C05474=1225.278,36.336,-43.631,-179.133,5.420,148.684
C05475=1225.283,36.087,-43.615,-179.135,5.420,148.685
C05476=1225.289,35.837,-43.599,-179.138,5.420,148.685
C05477=1225.293,35.588,-43.583,-179.141,5.419,148.686
C05478=1225.299,35.339,-43.567,-179.143,5.418,148.687
C05479=1225.304,35.088,-43.551,-179.146,5.418,148.687
C05480=1225.308,34.839,-43.536,-179.149,5.417,148.688
C05481=1225.313,34.591,-43.520,-179.151,5.417,148.689
C05482=1225.318,34.340,-43.504,-179.153,5.416,148.689
C05483=1225.323,34.091,-43.488,-179.156,5.416,148.690
C05484=1225.329,33.842,-43.472,-179.158,5.416,148.691
C05485=1225.333,33.592,-43.456,-179.161,5.415,148.691
C05486=1225.338,33.343,-43.441,-179.163,5.414,148.692
C05487=1225.343,33.093,-43.425,-179.166,5.414,148.693
C05488=1225.348,32.844,-43.410,-179.169,5.413,148.693
C05489=1225.353,32.595,-43.393,-179.171,5.413,148.694
C05490=1225.358,32.345,-43.377,-179.174,5.412,148.695
C05491=1225.363,32.096,-43.362,-179.176,5.413,148.695
C05492=1225.368,31.846,-43.347,-179.179,5.412,148.696
C05493=1225.373,31.596,-43.331,-179.181,5.411,148.697
C05494=1225.378,31.347,-43.314,-179.184,5.411,148.697
C05495=1225.383,31.098,-43.299,-179.186,5.410,148.698
C05496=1225.387,30.848,-43.284,-179.189,5.409,148.698
C05497=1225.393,30.599,-43.268,-179.191,5.409,148.699
C05498=1225.398,30.349,-43.252,-179.194,5.409,148.700
C05499=1225.403,30.099,-43.236,-179.196,5.409,148.701
C05500=1225.408,29.831,-43.220,-179.199,5.408,148.701
C05501=1225.413,29.563,-43.203,-179.201,5.408,148.702
C05502=1225.419,29.294,-43.186,-179.205,5.407,148.703
C05503=1225.424,29.026,-43.169,-179.207,5.407,148.703
C05504=1225.429,28.777,-43.154,-179.210,5.406,148.704
C05505=1225.434,28.526,-43.138,-179.213,5.406,148.705
C05506=1225.439,28.277,-43.122,-179.215,5.405,148.705
C05507=1225.445,28.028,-43.107,-179.217,5.404,148.706
C05508=1225.449,27.778,-43.091,-179.220,5.404,148.707
C05509=1225.454,27.528,-43.076,-179.222,5.404,148.707
C05510=1225.459,27.279,-43.060,-179.225,5.403,148.708
C05511=1225.464,27.030,-43.045,-179.227,5.403,148.709
C05512=1225.469,26.780,-43.029,-179.230,5.402,148.709
C05513=1225.474,26.530,-43.014,-179.233,5.402,148.710
C05514=1225.479,26.281,-42.999,-179.235,5.401,148.711
C05515=1225.484,26.032,-42.983,-179.237,5.401,148.711
C05516=1225.489,25.782,-42.967,-179.240,5.401,148.712
C05517=1225.494,25.533,-42.952,-179.243,5.400,148.713
C05518=1225.499,25.283,-42.937,-179.245,5.400,148.713
C05519=1225.504,25.034,-42.922,-179.248,5.399,148.714
C05520=1225.509,24.784,-42.906,-179.251,5.399,148.715
C05521=1225.514,24.535,-42.890,-179.253,5.398,148.715
C05522=1225.519,24.286,-42.875,-179.255,5.398,148.716
C05523=1225.524,24.036,-42.860,-179.257,5.398,148.717
C05524=1225.529,23.787,-42.844,-179.260,5.397,148.717
C05525=1225.533,23.537,-42.829,-179.263,5.397,148.718
C05526=1225.539,23.288,-42.813,-179.265,5.396,148.719
C05527=1225.544,23.038,-42.799,-179.268,5.395,148.719
C05528=1225.549,22.789,-42.783,-179.270,5.396,148.720
C05529=1225.553,22.539,-42.768,-179.273,5.395,148.721
C05530=1225.559,22.289,-42.752,-179.275,5.395,148.721
C05531=1225.564,22.040,-42.737,-179.278,5.394,148.722
C05532=1225.569,21.791,-42.722,-179.281,5.394,148.723
C05533=1225.574,21.541,-42.706,-179.283,5.394,148.723
C05534=1225.579,21.292,-42.691,-179.285,5.393,148.724
C05535=1225.584,21.042,-42.676,-179.288,5.393,148.725
C05536=1225.588,20.793,-42.661,-179.291,5.392,148.725
C05537=1225.594,20.543,-42.645,-179.293,5.392,148.726
C05538=1225.598,20.294,-42.630,-179.296,5.391,148.727
C05539=1225.604,20.045,-42.615,-179.298,5.391,148.727
C05540=1225.609,19.795,-42.600,-179.300,5.390,148.728
C05541=1225.614,19.545,-42.584,-179.303,5.390,148.729
C05542=1225.618,19.296,-42.569,-179.306,5.389,148.729
C05543=1225.624,19.046,-42.554,-179.308,5.389,148.730
C05544=1225.628,18.797,-42.539,-179.310,5.389,148.731
C05545=1225.634,18.547,-42.524,-179.313,5.389,148.731
C05546=1225.639,18.298,-42.509,-179.316,5.388,148.732
C05547=1225.644,18.049,-42.493,-179.318,5.388,148.733
C05548=1225.648,17.799,-42.478,-179.321,5.387,148.733
C05549=1225.654,17.549,-42.463,-179.323,5.386,148.734
C05550=1225.658,17.300,-42.448,-179.326,5.387,148.735
C05551=1225.664,17.050,-42.433,-179.328,5.386,148.735
C05552=1225.669,16.801,-42.418,-179.331,5.386,148.736
C05553=1225.674,16.551,-42.403,-179.334,5.385,148.737
C05554=1225.679,16.302,-42.388,-179.336,5.385,148.737
C05555=1225.683,16.053,-42.373,-179.338,5.385,148.738
C05556=1225.689,15.803,-42.358,-179.341,5.384,148.739
C05557=1225.693,15.553,-42.342,-179.344,5.384,148.740
C05558=1225.699,15.303,-42.328,-179.346,5.383,148.740
C05559=1225.703,15.054,-42.313,-179.349,5.383,148.741
C05560=1225.708,14.805,-42.298,-179.350,5.383,148.741
C05561=1225.714,14.555,-42.283,-179.353,5.382,148.742
C05562=1225.718,14.306,-42.268,-179.356,5.382,148.743
C05563=1225.724,14.057,-42.252,-179.358,5.381,148.743
C05564=1225.729,13.807,-42.238,-179.361,5.381,148.744
C05565=1225.733,13.558,-42.223,-179.363,5.381,148.745
C05566=1225.739,13.308,-42.208,-179.366,5.380,148.745
C05567=1225.744,13.059,-42.193,-179.368,5.380,148.746
C05568=1225.748,12.810,-42.178,-179.371,5.379,148.747
C05569=1225.754,12.560,-42.163,-179.373,5.379,148.748
C05570=1225.759,12.310,-42.148,-179.376,5.379,148.748
C05571=1225.764,12.060,-42.133,-179.378,5.378,148.749
C05572=1225.768,11.811,-42.118,-179.381,5.378,148.750
C05573=1225.773,11.561,-42.104,-179.384,5.377,148.750
C05574=1225.779,11.312,-42.088,-179.386,5.378,148.751
C05575=1225.784,11.062,-42.074,-179.388,5.377,148.752
C05576=1225.788,10.813,-42.059,-179.391,5.377,148.752
C05577=1225.793,10.563,-42.045,-179.394,5.376,148.753
C05578=1225.799,10.314,-42.029,-179.396,5.375,148.754
C05579=1225.804,10.064,-42.015,-179.398,5.376,148.754
C05580=1225.808,9.815,-42.000,-179.401,5.375,148.755
C05581=1225.814,9.565,-41.985,-179.404,5.375,148.756
C05582=1225.819,9.316,-41.970,-179.406,5.374,148.756
C05583=1225.824,9.066,-41.956,-179.408,5.374,148.757
C05584=1225.828,8.817,-41.941,-179.411,5.374,148.758
C05585=1225.834,8.567,-41.926,-179.414,5.373,148.759
C05586=1225.839,8.318,-41.911,-179.416,5.373,148.759
C05587=1225.844,8.068,-41.896,-179.418,5.373,148.760
C05588=1225.849,7.818,-41.882,-179.421,5.373,148.761
C05589=1225.854,7.569,-41.867,-179.424,5.372,148.761
C05590=1225.859,7.319,-41.852,-179.426,5.372,148.762
C05591=1225.864,7.070,-41.837,-179.429,5.371,148.762
C05592=1225.869,6.820,-41.823,-179.431,5.371,148.763
C05593=1225.874,6.570,-41.808,-179.433,5.370,148.764
C05594=1225.879,6.321,-41.793,-179.436,5.370,148.764
C05595=1225.884,6.072,-41.779,-179.439,5.369,148.765
C05596=1225.889,5.823,-41.764,-179.441,5.370,148.766
C05597=1225.894,5.574,-41.750,-179.443,5.369,148.767
C05598=1225.900,5.324,-41.735,-179.446,5.369,148.767
C05599=1225.904,5.074,-41.720,-179.449,5.368,148.768
C05600=1225.909,4.825,-41.706,-179.451,5.368,148.769
C05601=1225.914,4.575,-41.691,-179.453,5.368,148.769
C05602=1225.919,4.326,-41.677,-179.456,5.367,148.770
C05603=1225.924,4.076,-41.662,-179.459,5.367,148.771
C05604=1225.930,3.807,-41.646,-179.461,5.366,148.771
C05605=1225.935,3.538,-41.631,-179.464,5.367,148.772
C05606=1225.940,3.269,-41.615,-179.467,5.366,148.773
C05607=1225.945,3.000,-41.600,-179.469,5.366,148.774
C05608=1225.951,2.750,-41.585,-179.472,5.365,148.774
C05609=1225.956,2.501,-41.570,-179.475,5.365,148.775
C05610=1225.961,2.252,-41.556,-179.477,5.365,148.776
C05611=1225.966,2.002,-41.541,-179.479,5.365,148.776
C05612=1225.971,1.753,-41.527,-179.482,5.364,148.777
C05613=1225.976,1.503,-41.513,-179.485,5.364,148.778
C05614=1225.981,1.254,-41.498,-179.487,5.364,148.778
C05615=1225.986,1.004,-41.484,-179.489,5.363,148.779
C05616=1225.991,0.754,-41.469,-179.492,5.363,148.780
C05617=1225.996,0.505,-41.455,-179.495,5.362,148.781
C05618=1226.001,0.255,-41.440,-179.497,5.363,148.781
C05619=1226.007,0.006,-41.426,-179.499,5.362,148.782
C05620=1226.012,-0.243,-41.411,-179.502,5.362,148.783
C05621=1226.017,-0.493,-41.397,-179.505,5.361,148.783
C05622=1226.022,-0.743,-41.383,-179.507,5.361,148.784
C05623=1226.026,-0.993,-41.368,-179.509,5.361,148.785
C05624=1226.031,-1.242,-41.354,-179.512,5.360,148.785
C05625=1226.036,-1.492,-41.340,-179.515,5.360,148.786
C05626=1226.042,-1.740,-41.325,-179.517,5.360,148.787
C05627=1226.047,-1.990,-41.311,-179.519,5.359,148.787
C05628=1226.052,-2.240,-41.297,-179.522,5.359,148.788
C05629=1226.056,-2.490,-41.282,-179.525,5.358,148.789
C05630=1226.061,-2.739,-41.268,-179.527,5.359,148.789
C05631=1226.066,-2.989,-41.254,-179.529,5.358,148.790
C05632=1226.072,-3.238,-41.240,-179.532,5.358,148.791
C05633=1226.077,-3.488,-41.226,-179.534,5.358,148.792
C05634=1226.082,-3.737,-41.211,-179.537,5.357,148.792
C05635=1226.087,-3.987,-41.197,-179.539,5.357,148.793
C05636=1226.092,-4.237,-41.183,-179.542,5.356,148.794
C05637=1226.097,-4.486,-41.169,-179.544,5.357,148.794
C05638=1226.102,-4.736,-41.155,-179.547,5.356,148.795
C05639=1226.107,-4.985,-41.140,-179.550,5.356,148.796
C05640=1226.112,-5.235,-41.126,-179.552,5.355,148.796
C05641=1226.117,-5.485,-41.112,-179.554,5.355,148.797
C05642=1226.123,-5.734,-41.098,-179.557,5.355,148.798
C05643=1226.128,-5.983,-41.084,-179.560,5.354,148.798
C05644=1226.133,-6.233,-41.069,-179.562,5.355,148.799
C05645=1226.138,-6.483,-41.055,-179.564,5.354,148.800
C05646=1226.143,-6.733,-41.041,-179.567,5.354,148.801
C05647=1226.147,-6.981,-41.028,-179.570,5.353,148.801
C05648=1226.152,-7.231,-41.013,-179.572,5.353,148.802
C05649=1226.157,-7.481,-40.999,-179.574,5.353,148.803
C05650=1226.162,-7.730,-40.985,-179.577,5.352,148.803
C05651=1226.168,-7.979,-40.971,-179.579,5.353,148.804
C05652=1226.173,-8.229,-40.957,-179.582,5.352,148.805
C05653=1226.178,-8.479,-40.942,-179.584,5.352,148.805
C05654=1226.183,-8.729,-40.928,-179.587,5.351,148.806
C05655=1226.188,-8.978,-40.914,-179.589,5.352,148.807
C05656=1226.192,-9.227,-40.900,-179.592,5.351,148.807
C05657=1226.197,-9.477,-40.886,-179.594,5.350,148.808
C05658=1226.203,-9.727,-40.873,-179.597,5.351,148.809
C05659=1226.208,-9.976,-40.859,-179.599,5.350,148.810
C05660=1226.213,-10.226,-40.844,-179.602,5.350,148.810
C05661=1226.218,-10.475,-40.830,-179.604,5.350,148.811
C05662=1226.224,-10.724,-40.816,-179.607,5.350,148.812
C05663=1226.228,-10.974,-40.802,-179.609,5.349,148.812
C05664=1226.233,-11.224,-40.789,-179.612,5.349,148.813
C05665=1226.238,-11.474,-40.775,-179.614,5.349,148.814
C05666=1226.244,-11.723,-40.761,-179.617,5.348,148.814
C05667=1226.249,-11.973,-40.746,-179.619,5.348,148.815
C05668=1226.253,-12.222,-40.733,-179.621,5.348,148.816
C05669=1226.258,-12.471,-40.719,-179.624,5.348,148.816
C05670=1226.264,-12.721,-40.705,-179.627,5.347,148.817
C05671=1226.269,-12.971,-40.691,-179.629,5.347,148.818
C05672=1226.274,-13.220,-40.677,-179.631,5.347,148.819
C05673=1226.278,-13.469,-40.663,-179.634,5.346,148.819
C05674=1226.284,-13.720,-40.650,-179.637,5.346,148.820
C05675=1226.289,-13.969,-40.636,-179.639,5.346,148.821
C05676=1226.294,-14.218,-40.622,-179.641,5.346,148.821
C05677=1226.298,-14.468,-40.608,-179.644,5.345,148.822
C05678=1226.304,-14.717,-40.595,-179.646,5.345,148.823
C05679=1226.309,-14.967,-40.581,-179.649,5.345,148.823
C05680=1226.314,-15.217,-40.566,-179.651,5.344,148.824
C05681=1226.319,-15.466,-40.554,-179.654,5.345,148.825
C05682=1226.324,-15.716,-40.539,-179.656,5.344,148.825
C05683=1226.329,-15.966,-40.525,-179.659,5.344,148.826
C05684=1226.335,-16.215,-40.512,-179.661,5.344,148.827
C05685=1226.339,-16.465,-40.498,-179.664,5.343,148.828
C05686=1226.344,-16.714,-40.484,-179.666,5.343,148.828
C05687=1226.350,-16.964,-40.471,-179.668,5.343,148.829
C05688=1226.354,-17.213,-40.457,-179.671,5.343,148.830
C05689=1226.360,-17.462,-40.443,-179.674,5.342,148.830
C05690=1226.365,-17.713,-40.430,-179.676,5.342,148.831
C05691=1226.369,-17.962,-40.416,-179.678,5.342,148.832
C05692=1226.375,-18.211,-40.402,-179.681,5.342,148.832
C05693=1226.380,-18.462,-40.388,-179.684,5.341,148.833
C05694=1226.385,-18.711,-40.374,-179.686,5.341,148.834
C05695=1226.390,-18.961,-40.362,-179.688,5.341,148.834
C05696=1226.395,-19.210,-40.347,-179.691,5.340,148.835
C05697=1226.400,-19.459,-40.334,-179.693,5.341,148.836
C05698=1226.405,-19.709,-40.320,-179.696,5.340,148.837
C05699=1226.411,-19.958,-40.306,-179.699,5.340,148.837
C05700=1226.415,-20.208,-40.294,-179.701,5.340,148.838
C05701=1226.420,-20.458,-40.279,-179.703,5.339,148.839
C05702=1226.426,-20.708,-40.266,-179.706,5.339,148.839
C05703=1226.430,-20.957,-40.252,-179.708,5.339,148.840
C05704=1226.436,-21.207,-40.239,-179.711,5.339,148.841
C05705=1226.441,-21.456,-40.225,-179.713,5.338,148.841
C05706=1226.446,-21.706,-40.212,-179.715,5.339,148.842
C05707=1226.451,-21.955,-40.198,-179.718,5.338,148.843
C05708=1226.457,-22.225,-40.183,-179.721,5.338,148.844
C05709=1226.462,-22.494,-40.170,-179.723,5.337,148.844
C05710=1226.468,-22.763,-40.155,-179.726,5.338,148.845
C05711=1226.473,-23.033,-40.140,-179.729,5.337,148.846
C05712=1226.478,-23.282,-40.127,-179.731,5.337,148.847
C05713=1226.483,-23.532,-40.113,-179.733,5.337,148.847
C05714=1226.488,-23.782,-40.100,-179.736,5.336,148.848
C05715=1226.493,-24.031,-40.086,-179.739,5.336,148.849
C05716=1226.498,-24.281,-40.073,-179.741,5.336,148.849
C05717=1226.503,-24.530,-40.059,-179.743,5.336,148.850
C05718=1226.509,-24.780,-40.046,-179.746,5.335,148.851
C05719=1226.514,-25.029,-40.033,-179.748,5.336,148.851
C05720=1226.519,-25.279,-40.019,-179.751,5.335,148.852
C05721=1226.524,-25.528,-40.006,-179.753,5.335,148.853
C05722=1226.529,-25.778,-39.992,-179.756,5.335,148.853
C05723=1226.534,-26.027,-39.979,-179.758,5.334,148.854
C05724=1226.539,-26.278,-39.966,-179.761,5.334,148.855
C05725=1226.544,-26.526,-39.952,-179.763,5.334,148.856
C05726=1226.549,-26.777,-39.939,-179.766,5.334,148.856
C05727=1226.554,-27.026,-39.926,-179.768,5.333,148.857
C05728=1226.559,-27.276,-39.912,-179.770,5.334,148.858
C05729=1226.564,-27.525,-39.899,-179.773,5.333,148.858
C05730=1226.570,-27.775,-39.886,-179.776,5.333,148.859
C05731=1226.575,-28.024,-39.872,-179.778,5.333,148.860
C05732=1226.579,-28.274,-39.859,-179.780,5.332,148.860
C05733=1226.585,-28.524,-39.846,-179.783,5.333,148.861
C05734=1226.589,-28.773,-39.833,-179.785,5.332,148.862
C05735=1226.595,-29.023,-39.819,-179.788,5.332,148.863
C05736=1226.600,-29.272,-39.807,-179.790,5.332,148.863
C05737=1226.605,-29.522,-39.792,-179.793,5.331,148.864
C05738=1226.610,-29.771,-39.780,-179.795,5.331,148.865
C05739=1226.615,-30.022,-39.766,-179.797,5.331,148.865
C05740=1226.621,-30.271,-39.754,-179.800,5.331,148.866
C05741=1226.625,-30.520,-39.740,-179.803,5.330,148.867
C05742=1226.631,-30.770,-39.727,-179.805,5.331,148.867
C05743=1226.635,-31.020,-39.714,-179.807,5.330,148.868
C05744=1226.641,-31.270,-39.701,-179.809,5.330,148.869
C05745=1226.646,-31.519,-39.688,-179.812,5.330,148.870
C05746=1226.650,-31.768,-39.674,-179.815,5.329,148.870
C05747=1226.656,-32.018,-39.661,-179.817,5.330,148.871
C05748=1226.661,-32.268,-39.648,-179.820,5.329,148.872
C05749=1226.666,-32.517,-39.636,-179.822,5.329,148.872
C05750=1226.672,-32.767,-39.622,-179.824,5.329,148.873
C05751=1226.676,-33.016,-39.609,-179.827,5.329,148.874
C05752=1226.682,-33.266,-39.596,-179.830,5.328,148.874
C05753=1226.686,-33.516,-39.583,-179.832,5.328,148.875
C05754=1226.691,-33.765,-39.570,-179.834,5.328,148.876
C05755=1226.697,-34.015,-39.557,-179.837,5.329,148.877
C05756=1226.702,-34.265,-39.544,-179.840,5.328,148.877
C05757=1226.707,-34.514,-39.531,-179.842,5.328,148.878
C05758=1226.712,-34.764,-39.517,-179.844,5.328,148.879
C05759=1226.717,-35.013,-39.504,-179.847,5.327,148.880
C05760=1226.722,-35.263,-39.492,-179.850,5.327,148.880
C05761=1226.727,-35.513,-39.478,-179.852,5.327,148.881
C05762=1226.733,-35.762,-39.466,-179.854,5.327,148.882
C05763=1226.738,-36.011,-39.453,-179.856,5.327,148.882
C05764=1226.742,-36.262,-39.440,-179.859,5.327,148.883
C05765=1226.748,-36.511,-39.427,-179.862,5.326,148.884
C05766=1226.753,-36.760,-39.414,-179.864,5.326,148.884
C05767=1226.758,-37.010,-39.401,-179.867,5.326,148.885
C05768=1226.764,-37.260,-39.388,-179.869,5.325,148.886
C05769=1226.769,-37.509,-39.375,-179.871,5.326,148.887
C05770=1226.773,-37.759,-39.362,-179.874,5.325,148.887
C05771=1226.778,-38.009,-39.350,-179.876,5.326,148.888
C05772=1226.784,-38.258,-39.337,-179.879,5.325,148.889
C05773=1226.789,-38.508,-39.324,-179.881,5.325,148.889
C05774=1226.794,-38.758,-39.311,-179.883,5.325,148.890
C05775=1226.799,-39.007,-39.298,-179.886,5.324,148.891
C05776=1226.804,-39.257,-39.285,-179.888,5.325,148.891
C05777=1226.809,-39.507,-39.272,-179.891,5.324,148.892
C05778=1226.814,-39.756,-39.260,-179.894,5.324,148.893
C05779=1226.819,-40.006,-39.247,-179.896,5.324,148.894
C05780=1226.824,-40.255,-39.234,-179.898,5.324,148.894
C05781=1226.830,-40.505,-39.221,-179.901,5.323,148.895
C05782=1226.835,-40.754,-39.208,-179.903,5.323,148.896
C05783=1226.840,-41.004,-39.195,-179.906,5.323,148.896
C05784=1226.845,-41.254,-39.183,-179.908,5.323,148.897
C05785=1226.850,-41.503,-39.170,-179.910,5.323,148.898
C05786=1226.855,-41.753,-39.157,-179.913,5.322,148.898
C05787=1226.860,-42.003,-39.144,-179.915,5.323,148.899
C05788=1226.865,-42.252,-39.131,-179.918,5.322,148.900
C05789=1226.871,-42.501,-39.119,-179.920,5.322,148.901
C05790=1226.875,-42.751,-39.106,-179.923,5.322,148.901
C05791=1226.880,-43.001,-39.094,-179.925,5.321,148.902
C05792=1226.886,-43.251,-39.081,-179.927,5.322,148.903
C05793=1226.891,-43.501,-39.068,-179.930,5.321,148.903
C05794=1226.896,-43.750,-39.055,-179.932,5.322,148.904
C05795=1226.901,-43.999,-39.043,-179.935,5.321,148.905
C05796=1226.906,-44.249,-39.030,-179.937,5.321,148.905
C05797=1226.911,-44.499,-39.017,-179.940,5.321,148.906
C05798=1226.916,-44.749,-39.005,-179.942,5.321,148.907
C05799=1226.921,-44.998,-38.993,-179.944,5.321,148.908
C05800=1226.927,-45.248,-38.979,-179.947,5.320,148.908
C05801=1226.932,-45.497,-38.967,-179.950,5.320,148.909
C05802=1226.937,-45.747,-38.954,-179.952,5.320,148.910
C05803=1226.942,-45.997,-38.942,-179.954,5.320,148.910
C05804=1226.947,-46.246,-38.929,-179.956,5.320,148.911
C05805=1226.952,-46.496,-38.917,-179.959,5.320,148.912
C05806=1226.957,-46.746,-38.904,-179.962,5.319,148.912
C05807=1226.962,-46.996,-38.892,-179.964,5.319,148.913
C05808=1226.968,-47.245,-38.879,-179.967,5.319,148.914
C05809=1226.973,-47.494,-38.867,-179.969,5.319,148.915
C05810=1226.978,-47.743,-38.854,-179.971,5.319,148.915
C05811=1226.983,-47.994,-38.842,-179.973,5.319,148.916
C05812=1226.989,-48.263,-38.828,-179.977,5.319,148.917
C05813=1226.994,-48.533,-38.814,-179.979,5.319,148.918
C05814=1227.000,-48.803,-38.802,-179.982,5.318,148.918
C05815=1227.006,-49.073,-38.787,-179.984,5.318,148.919
C05816=1227.011,-49.322,-38.775,-179.987,5.318,148.920
C05817=1227.016,-49.573,-38.762,-179.989,5.318,148.920
C05818=1227.021,-49.822,-38.750,-179.991,5.318,148.921
C05819=1227.026,-50.071,-38.737,-179.994,5.317,148.922
C05820=1227.031,-50.321,-38.725,-179.996,5.318,148.923
C05821=1227.036,-50.571,-38.713,-179.999,5.317,148.923
C05822=1227.042,-50.820,-38.700,179.999,5.317,148.924
C05823=1227.047,-51.070,-38.688,179.996,5.317,148.925
C05824=1227.051,-51.320,-38.675,179.994,5.316,148.925
C05825=1227.057,-51.569,-38.663,179.992,5.317,148.926
C05826=1227.062,-51.819,-38.651,179.989,5.316,148.927
C05827=1227.067,-52.069,-38.638,179.987,5.317,148.927
C05828=1227.072,-52.318,-38.626,179.984,5.316,148.928
C05829=1227.077,-52.568,-38.614,179.982,5.316,148.929
C05830=1227.082,-52.817,-38.602,179.980,5.316,148.930
C05831=1227.087,-53.067,-38.590,179.977,5.316,148.930
C05832=1227.092,-53.317,-38.577,179.975,5.316,148.931
C05833=1227.097,-53.566,-38.564,179.972,5.315,148.932
C05834=1227.103,-53.816,-38.552,179.970,5.316,148.933
C05835=1227.108,-54.065,-38.540,179.967,5.316,148.933
C05836=1227.113,-54.315,-38.528,179.965,5.316,148.934
C05837=1227.118,-54.565,-38.515,179.962,5.315,148.935
C05838=1227.124,-54.815,-38.503,179.959,5.315,148.935
C05839=1227.128,-55.065,-38.490,179.957,5.315,148.936
C05840=1227.133,-55.314,-38.479,179.955,5.315,148.937
C05841=1227.138,-55.564,-38.467,179.953,5.315,148.938
C05842=1227.143,-55.813,-38.455,179.950,5.315,148.938
C05843=1227.149,-56.063,-38.442,179.948,5.315,148.939
C05844=1227.154,-56.313,-38.430,179.945,5.315,148.940
C05845=1227.159,-56.562,-38.418,179.943,5.314,148.940
C05846=1227.165,-56.812,-38.406,179.940,5.314,148.941
C05847=1227.170,-57.061,-38.393,179.938,5.314,148.942
C05848=1227.174,-57.311,-38.382,179.936,5.314,148.943
C05849=1227.180,-57.560,-38.369,179.933,5.314,148.943
C05850=1227.185,-57.810,-38.357,179.931,5.314,148.944
C05851=1227.189,-58.060,-38.344,179.928,5.314,148.945
C05852=1227.195,-58.310,-38.333,179.926,5.313,148.945
C05853=1227.200,-58.560,-38.321,179.924,5.314,148.946
C05854=1227.205,-58.809,-38.309,179.921,5.313,148.947
C05855=1227.210,-59.059,-38.297,179.919,5.313,148.947
C05856=1227.215,-59.308,-38.284,179.916,5.313,148.948
C05857=1227.221,-59.558,-38.272,179.914,5.313,148.949
C05858=1227.226,-59.808,-38.260,179.911,5.313,148.950
C05859=1227.231,-60.057,-38.248,179.909,5.313,148.950
C05860=1227.236,-60.307,-38.236,179.907,5.313,148.951
C05861=1227.241,-60.556,-38.224,179.904,5.312,148.952
C05862=1227.246,-60.806,-38.212,179.902,5.313,148.952
C05863=1227.251,-61.056,-38.201,179.899,5.312,148.953
C05864=1227.256,-61.305,-38.188,179.897,5.312,148.954
C05865=1227.262,-61.555,-38.176,179.894,5.312,148.954
C05866=1227.267,-61.805,-38.164,179.892,5.312,148.955
C05867=1227.272,-62.055,-38.152,179.890,5.312,148.956
C05868=1227.277,-62.304,-38.140,179.888,5.312,148.957
C05869=1227.282,-62.554,-38.129,179.885,5.312,148.957
C05870=1227.288,-62.803,-38.116,179.882,5.311,148.958
C05871=1227.293,-63.053,-38.104,179.880,5.312,148.959
C05872=1227.298,-63.303,-38.093,179.877,5.311,148.959
C05873=1227.303,-63.552,-38.080,179.875,5.311,148.960
C05874=1227.308,-63.802,-38.068,179.873,5.311,148.961
C05875=1227.313,-64.052,-38.057,179.871,5.311,148.962
C05876=1227.318,-64.302,-38.045,179.868,5.311,148.962
C05877=1227.323,-64.551,-38.033,179.866,5.311,148.963
C05878=1227.329,-64.801,-38.021,179.863,5.311,148.964
C05879=1227.334,-65.051,-38.009,179.861,5.311,148.964
C05880=1227.339,-65.301,-37.997,179.858,5.311,148.965
C05881=1227.344,-65.550,-37.985,179.856,5.310,148.966
C05882=1227.349,-65.800,-37.974,179.854,5.310,148.966
C05883=1227.354,-66.049,-37.962,179.851,5.310,148.967
C05884=1227.360,-66.299,-37.950,179.849,5.310,148.968
C05885=1227.365,-66.548,-37.939,179.846,5.310,148.969
C05886=1227.370,-66.798,-37.926,179.844,5.310,148.969
C05887=1227.376,-67.048,-37.914,179.842,5.310,148.970
C05888=1227.380,-67.297,-37.903,179.839,5.310,148.971
C05889=1227.386,-67.547,-37.891,179.837,5.310,148.971
C05890=1227.391,-67.797,-37.879,179.835,5.310,148.972
C05891=1227.395,-68.046,-37.867,179.832,5.309,148.973
C05892=1227.401,-68.296,-37.855,179.829,5.309,148.974
C05893=1227.406,-68.546,-37.844,179.827,5.309,148.974
C05894=1227.411,-68.796,-37.832,179.825,5.309,148.975
C05895=1227.416,-69.046,-37.820,179.822,5.309,148.976
C05896=1227.421,-69.295,-37.809,179.820,5.309,148.976
C05897=1227.427,-69.544,-37.798,179.818,5.309,148.977
C05898=1227.433,-69.794,-37.786,179.815,5.309,148.978
C05899=1227.437,-70.043,-37.774,179.813,5.309,148.979
C05900=1227.442,-70.293,-37.762,179.810,5.308,148.979
C05901=1227.447,-70.543,-37.750,179.808,5.309,148.980
C05902=1227.453,-70.793,-37.739,179.806,5.308,148.980
C05903=1227.457,-71.042,-37.727,179.804,5.308,148.981
C05904=1227.463,-71.292,-37.715,179.801,5.308,148.982
C05905=1227.468,-71.542,-37.704,179.799,5.308,148.983
C05906=1227.473,-71.791,-37.693,179.797,5.308,148.983
C05907=1227.479,-72.041,-37.681,179.794,5.307,148.984
C05908=1227.483,-72.291,-37.669,179.792,5.308,148.985
C05909=1227.489,-72.541,-37.658,179.789,5.307,148.985
C05910=1227.494,-72.790,-37.646,179.787,5.307,148.986
C05911=1227.499,-73.040,-37.634,179.784,5.307,148.987
C05912=1227.504,-73.290,-37.623,179.782,5.307,148.987
C05913=1227.510,-73.539,-37.612,179.780,5.307,148.988
C05914=1227.515,-73.789,-37.600,179.777,5.307,148.989
C05915=1227.520,-74.039,-37.588,179.775,5.307,148.990
C05916=1227.525,-74.309,-37.575,179.772,5.308,148.991
C05917=1227.531,-74.579,-37.564,179.770,5.307,148.991
C05918=1227.537,-74.850,-37.551,179.767,5.307,148.992
C05919=1227.542,-75.121,-37.538,179.765,5.307,148.993
C05920=1227.548,-75.370,-37.527,179.762,5.307,148.993
C05921=1227.553,-75.620,-37.516,179.760,5.307,148.994
C05922=1227.558,-75.869,-37.504,179.757,5.306,148.995
C05923=1227.563,-76.119,-37.492,179.755,5.307,148.996
C05924=1227.568,-76.369,-37.481,179.753,5.306,148.996
C05925=1227.574,-76.618,-37.470,179.750,5.306,148.997
C05926=1227.579,-76.868,-37.458,179.748,5.306,148.998
C05927=1227.584,-77.118,-37.446,179.745,5.306,148.998
C05928=1227.589,-77.367,-37.435,179.743,5.306,148.999
C05929=1227.594,-77.617,-37.423,179.740,5.306,149.000
C05930=1227.600,-77.867,-37.413,179.738,5.306,149.000
C05931=1227.604,-78.116,-37.402,179.736,5.305,149.001
C05932=1227.610,-78.366,-37.390,179.734,5.306,149.002
C05933=1227.615,-78.616,-37.379,179.731,5.305,149.003
C05934=1227.620,-78.866,-37.367,179.729,5.306,149.003
C05935=1227.625,-79.115,-37.356,179.726,5.305,149.004
C05936=1227.630,-79.364,-37.344,179.724,5.306,149.005
C05937=1227.636,-79.615,-37.333,179.721,5.305,149.005
C05938=1227.640,-79.865,-37.322,179.719,5.306,149.006
C05939=1227.646,-80.114,-37.310,179.717,5.305,149.007
C05940=1227.651,-80.363,-37.299,179.714,5.305,149.008
C05941=1227.656,-80.613,-37.288,179.712,5.305,149.008
C05942=1227.662,-80.864,-37.277,179.710,5.305,149.009
C05943=1227.667,-81.112,-37.266,179.707,5.305,149.010
C05944=1227.672,-81.362,-37.254,179.705,5.305,149.010
C05945=1227.677,-81.612,-37.243,179.702,5.305,149.011
C05946=1227.682,-81.862,-37.231,179.700,5.305,149.012
C05947=1227.688,-82.112,-37.220,179.698,5.305,149.013
C05948=1227.693,-82.361,-37.209,179.695,5.305,149.013
C05949=1227.697,-82.611,-37.198,179.693,5.304,149.014
C05950=1227.703,-82.860,-37.186,179.691,5.305,149.014
C05951=1227.708,-83.110,-37.176,179.689,5.304,149.015
C05952=1227.713,-83.360,-37.165,179.686,5.304,149.016
C05953=1227.719,-83.610,-37.153,179.684,5.304,149.017
C05954=1227.724,-83.859,-37.142,179.682,5.304,149.017
C05955=1227.729,-84.109,-37.131,179.679,5.304,149.018
C05956=1227.734,-84.359,-37.119,179.677,5.304,149.019
C05957=1227.740,-84.608,-37.108,179.674,5.304,149.019
C05958=1227.745,-84.858,-37.098,179.672,5.304,149.020
C05959=1227.749,-85.108,-37.086,179.669,5.304,149.021
C05960=1227.755,-85.358,-37.075,179.667,5.304,149.022
C05961=1227.760,-85.607,-37.064,179.665,5.304,149.022
C05962=1227.765,-85.857,-37.053,179.663,5.304,149.023
C05963=1227.770,-86.106,-37.042,179.660,5.303,149.024
C05964=1227.776,-86.356,-37.031,179.658,5.304,149.024
C05965=1227.781,-86.606,-37.020,179.655,5.303,149.025
C05966=1227.785,-86.856,-37.008,179.653,5.304,149.026
C05967=1227.792,-87.105,-36.998,179.650,5.303,149.027
C05968=1227.796,-87.355,-36.986,179.648,5.304,149.027
C05969=1227.801,-87.605,-36.975,179.646,5.303,149.028
C05970=1227.807,-87.854,-36.965,179.644,5.304,149.029
C05971=1227.811,-88.104,-36.954,179.641,5.303,149.029
C05972=1227.817,-88.354,-36.942,179.639,5.303,149.030
C05973=1227.822,-88.603,-36.931,179.636,5.303,149.031
C05974=1227.827,-88.854,-36.921,179.634,5.303,149.031
C05975=1227.832,-89.103,-36.910,179.632,5.303,149.032
C05976=1227.838,-89.352,-36.898,179.630,5.303,149.033
C05977=1227.843,-89.603,-36.887,179.627,5.302,149.033
C05978=1227.848,-89.852,-36.877,179.625,5.303,149.034
C05979=1227.853,-90.102,-36.866,179.622,5.302,149.035
C05980=1227.858,-90.351,-36.855,179.620,5.303,149.036
C05981=1227.864,-90.601,-36.844,179.618,5.302,149.036
C05982=1227.869,-90.851,-36.833,179.615,5.303,149.037
C05983=1227.874,-91.101,-36.822,179.613,5.302,149.038
C05984=1227.879,-91.350,-36.811,179.611,5.303,149.038
C05985=1227.884,-91.600,-36.801,179.608,5.302,149.039
C05986=1227.890,-91.849,-36.790,179.606,5.302,149.040
C05987=1227.895,-92.100,-36.778,179.603,5.302,149.041
C05988=1227.900,-92.349,-36.767,179.601,5.302,149.041
C05989=1227.906,-92.599,-36.757,179.598,5.302,149.042
C05990=1227.910,-92.849,-36.746,179.596,5.302,149.043
C05991=1227.916,-93.098,-36.735,179.594,5.302,149.043
C05992=1227.921,-93.348,-36.724,179.592,5.302,149.044
C05993=1227.926,-93.597,-36.714,179.589,5.302,149.045
C05994=1227.931,-93.847,-36.703,179.587,5.302,149.045
C05995=1227.937,-94.098,-36.691,179.585,5.301,149.046
C05996=1227.942,-94.347,-36.681,179.583,5.302,149.047
C05997=1227.947,-94.597,-36.670,179.580,5.301,149.047
C05998=1227.953,-94.846,-36.660,179.578,5.302,149.048
C05999=1227.957,-95.096,-36.648,179.575,5.301,149.049
C06000=1227.963,-95.345,-36.638,179.573,5.301,149.050
C06001=1227.968,-95.596,-36.628,179.570,5.301,149.050
C06002=1227.973,-95.845,-36.616,179.568,5.301,149.051
C06003=1227.978,-96.095,-36.606,179.566,5.301,149.052
C06004=1227.983,-96.344,-36.595,179.564,5.301,149.052
C06005=1227.989,-96.594,-36.584,179.561,5.301,149.053
C06006=1227.994,-96.845,-36.574,179.559,5.301,149.054
C06007=1228.000,-97.093,-36.563,179.556,5.301,149.055
C06008=1228.005,-97.344,-36.552,179.554,5.301,149.055
C06009=1228.010,-97.593,-36.542,179.551,5.301,149.056
C06010=1228.015,-97.843,-36.531,179.550,5.301,149.056
C06011=1228.020,-98.092,-36.520,179.548,5.301,149.057
C06012=1228.025,-98.343,-36.510,179.545,5.301,149.058
C06013=1228.031,-98.592,-36.499,179.543,5.301,149.059
C06014=1228.036,-98.842,-36.488,179.540,5.301,149.059
C06015=1228.041,-99.091,-36.478,179.538,5.301,149.060
C06016=1228.046,-99.341,-36.467,179.535,5.300,149.061
C06017=1228.052,-99.591,-36.457,179.533,5.301,149.061
C06018=1228.057,-99.841,-36.446,179.531,5.300,149.062
C06019=1228.062,-100.090,-36.436,179.529,5.301,149.063
C06020=1228.067,-100.361,-36.424,179.526,5.300,149.064
C06021=1228.073,-100.633,-36.413,179.523,5.300,149.064
C06022=1228.079,-100.903,-36.401,179.521,5.300,149.065
C06023=1228.084,-101.174,-36.390,179.518,5.300,149.066
C06024=1228.089,-101.424,-36.379,179.516,5.300,149.066
C06025=1228.095,-101.673,-36.368,179.514,5.300,149.067
C06026=1228.100,-101.924,-36.358,179.512,5.300,149.068
C06027=1228.105,-102.173,-36.347,179.509,5.300,149.069
C06028=1228.110,-102.423,-36.337,179.507,5.300,149.069
C06029=1228.116,-102.673,-36.327,179.504,5.300,149.070
C06030=1228.121,-102.922,-36.316,179.502,5.300,149.071
C06031=1228.126,-103.172,-36.305,179.499,5.299,149.071
C06032=1228.132,-103.422,-36.295,179.497,5.300,149.072
C06033=1228.137,-103.672,-36.284,179.495,5.300,149.073
C06034=1228.142,-103.921,-36.275,179.492,5.300,149.074
C06035=1228.147,-104.171,-36.264,179.490,5.300,149.074
C06036=1228.152,-104.420,-36.253,179.488,5.299,149.075
C06037=1228.157,-104.671,-36.243,179.486,5.300,149.075
C06038=1228.162,-104.920,-36.232,179.483,5.299,149.076
C06039=1228.168,-105.170,-36.222,179.481,5.300,149.077
C06040=1228.173,-105.420,-36.212,179.479,5.299,149.078
C06041=1228.179,-105.669,-36.202,179.477,5.300,149.078
C06042=1228.184,-105.920,-36.191,179.474,5.299,149.079
C06043=1228.189,-106.169,-36.180,179.472,5.299,149.080
C06044=1228.193,-106.418,-36.170,179.469,5.299,149.080
C06045=1228.199,-106.668,-36.160,179.467,5.299,149.081
C06046=1228.204,-106.918,-36.150,179.464,5.299,149.082
C06047=1228.209,-107.168,-36.139,179.463,5.299,149.082
C06048=1228.215,-107.417,-36.129,179.460,5.299,149.083
C06049=1228.220,-107.668,-36.118,179.458,5.299,149.084
C06050=1228.226,-107.917,-36.108,179.456,5.299,149.085
C06051=1228.230,-108.166,-36.098,179.453,5.299,149.085
C06052=1228.235,-108.417,-36.088,179.451,5.299,149.086
C06053=1228.241,-108.666,-36.078,179.448,5.299,149.087
C06054=1228.247,-108.916,-36.067,179.446,5.299,149.087
C06055=1228.252,-109.166,-36.057,179.444,5.299,149.088
C06056=1228.257,-109.415,-36.047,179.442,5.299,149.089
C06057=1228.262,-109.665,-36.037,179.439,5.298,149.089
C06058=1228.267,-109.915,-36.026,179.437,5.299,149.090
C06059=1228.273,-110.165,-36.016,179.435,5.298,149.091
C06060=1228.278,-110.415,-36.006,179.433,5.299,149.091
C06061=1228.283,-110.664,-35.996,179.430,5.298,149.092
C06062=1228.288,-110.914,-35.986,179.428,5.299,149.093
C06063=1228.293,-111.164,-35.975,179.426,5.299,149.094
C06064=1228.299,-111.413,-35.965,179.423,5.298,149.094
C06065=1228.304,-111.663,-35.955,179.421,5.299,149.095
C06066=1228.309,-111.913,-35.945,179.419,5.298,149.095
C06067=1228.314,-112.162,-35.935,179.417,5.298,149.096
C06068=1228.320,-112.412,-35.924,179.414,5.298,149.097
C06069=1228.325,-112.662,-35.914,179.412,5.298,149.098
C06070=1228.330,-112.911,-35.904,179.409,5.298,149.098
C06071=1228.335,-113.161,-35.894,179.407,5.298,149.099
C06072=1228.340,-113.411,-35.884,179.404,5.298,149.100
C06073=1228.346,-113.661,-35.873,179.402,5.298,149.101
C06074=1228.351,-113.911,-35.864,179.400,5.298,149.101
C06075=1228.356,-114.161,-35.854,179.398,5.298,149.102
C06076=1228.362,-114.410,-35.844,179.396,5.298,149.102
C06077=1228.367,-114.660,-35.833,179.393,5.298,149.103
C06078=1228.372,-114.910,-35.823,179.391,5.298,149.104
C06079=1228.377,-115.159,-35.813,179.388,5.298,149.105
C06080=1228.383,-115.409,-35.803,179.386,5.298,149.105
C06081=1228.388,-115.658,-35.793,179.384,5.298,149.106
C06082=1228.393,-115.909,-35.784,179.382,5.298,149.107
C06083=1228.398,-116.159,-35.773,179.379,5.297,149.107
C06084=1228.403,-116.408,-35.764,179.377,5.298,149.108
C06085=1228.408,-116.658,-35.753,179.375,5.297,149.109
C06086=1228.414,-116.908,-35.743,179.373,5.297,149.109
C06087=1228.419,-117.157,-35.733,179.370,5.298,149.110
C06088=1228.425,-117.407,-35.724,179.368,5.297,149.111
C06089=1228.430,-117.657,-35.713,179.366,5.298,149.111
C06090=1228.435,-117.906,-35.704,179.363,5.297,149.112
C06091=1228.440,-118.156,-35.693,179.361,5.297,149.113
C06092=1228.446,-118.406,-35.683,179.359,5.297,149.113
C06093=1228.450,-118.656,-35.674,179.357,5.297,149.114
C06094=1228.456,-118.906,-35.664,179.354,5.297,149.115
C06095=1228.462,-119.155,-35.654,179.352,5.297,149.116
C06096=1228.466,-119.404,-35.644,179.349,5.297,149.116
C06097=1228.472,-119.655,-35.634,179.347,5.297,149.117
C06098=1228.477,-119.904,-35.624,179.345,5.297,149.117
C06099=1228.482,-120.154,-35.614,179.343,5.297,149.118
C06100=1228.488,-120.404,-35.604,179.341,5.297,149.119
C06101=1228.492,-120.654,-35.595,179.338,5.297,149.120
C06102=1228.498,-120.904,-35.585,179.336,5.297,149.120
C06103=1228.503,-121.153,-35.575,179.333,5.297,149.121
C06104=1228.509,-121.403,-35.565,179.331,5.297,149.122
C06105=1228.514,-121.653,-35.555,179.329,5.296,149.122
C06106=1228.519,-121.903,-35.545,179.327,5.297,149.123
C06107=1228.524,-122.153,-35.536,179.325,5.297,149.124
C06108=1228.529,-122.402,-35.526,179.322,5.297,149.124
C06109=1228.535,-122.651,-35.516,179.320,5.297,149.125
C06110=1228.540,-122.901,-35.507,179.317,5.297,149.126
C06111=1228.545,-123.152,-35.496,179.316,5.297,149.126
C06112=1228.550,-123.401,-35.487,179.313,5.296,149.127
C06113=1228.556,-123.651,-35.477,179.311,5.297,149.128
C06114=1228.561,-123.901,-35.467,179.308,5.296,149.128
C06115=1228.566,-124.150,-35.458,179.306,5.296,149.129
C06116=1228.572,-124.401,-35.448,179.303,5.296,149.130
C06117=1228.576,-124.650,-35.438,179.301,5.296,149.131
C06118=1228.582,-124.900,-35.429,179.300,5.296,149.131
C06119=1228.587,-125.149,-35.419,179.297,5.296,149.132
C06120=1228.593,-125.399,-35.409,179.295,5.296,149.133
C06121=1228.598,-125.649,-35.400,179.292,5.296,149.133
C06122=1228.603,-125.899,-35.389,179.290,5.296,149.134
C06123=1228.608,-126.149,-35.380,179.288,5.296,149.135
C06124=1228.186,-126.159,-35.416,179.284,5.299,149.137
C06125=1228.181,-125.910,-35.426,179.286,5.300,149.136
C06126=1228.177,-125.659,-35.435,179.288,5.299,149.135
C06127=1228.171,-125.410,-35.445,179.291,5.300,149.135
C06128=1228.166,-125.160,-35.455,179.293,5.300,149.134
C06129=1228.160,-124.910,-35.464,179.295,5.300,149.133
C06130=1228.155,-124.661,-35.474,179.297,5.300,149.133
C06131=1228.150,-124.411,-35.483,179.300,5.299,149.132
C06132=1228.144,-124.161,-35.494,179.302,5.300,149.131
C06133=1228.140,-123.911,-35.504,179.304,5.300,149.131
C06134=1228.134,-123.661,-35.513,179.306,5.300,149.130
C06135=1228.129,-123.412,-35.523,179.309,5.300,149.129
C06136=1228.123,-123.162,-35.533,179.311,5.300,149.128
C06137=1228.118,-122.912,-35.542,179.313,5.300,149.128
C06138=1228.113,-122.662,-35.552,179.316,5.300,149.127
C06139=1228.108,-122.412,-35.561,179.318,5.300,149.127
C06140=1228.102,-122.163,-35.571,179.320,5.300,149.126
C06141=1228.097,-121.914,-35.581,179.322,5.300,149.125
C06142=1228.092,-121.663,-35.591,179.324,5.300,149.124
C06143=1228.087,-121.413,-35.601,179.327,5.300,149.124
C06144=1228.082,-121.164,-35.611,179.329,5.300,149.123
C06145=1228.076,-120.914,-35.621,179.332,5.300,149.122
C06146=1228.071,-120.665,-35.630,179.334,5.300,149.122
C06147=1228.066,-120.414,-35.640,179.336,5.301,149.121
C06148=1228.060,-120.165,-35.651,179.338,5.300,149.120
C06149=1228.055,-119.915,-35.659,179.341,5.301,149.120
C06150=1228.050,-119.665,-35.670,179.343,5.300,149.119
C06151=1228.045,-119.416,-35.679,179.345,5.300,149.118
C06152=1228.040,-119.166,-35.690,179.348,5.300,149.117
C06153=1228.034,-118.916,-35.699,179.349,5.300,149.117
C06154=1228.029,-118.667,-35.709,179.352,5.301,149.116
C06155=1228.023,-118.417,-35.719,179.354,5.300,149.116
C06156=1228.019,-118.167,-35.729,179.357,5.301,149.115
C06157=1228.013,-117.917,-35.739,179.359,5.301,149.114
C06158=1228.008,-117.667,-35.749,179.362,5.301,149.113
C06159=1228.003,-117.418,-35.759,179.364,5.301,149.113
C06160=1227.998,-117.168,-35.769,179.365,5.301,149.112
C06161=1227.992,-116.918,-35.779,179.368,5.301,149.111
C06162=1227.987,-116.668,-35.788,179.370,5.301,149.111
C06163=1227.982,-116.418,-35.799,179.373,5.301,149.110
C06164=1227.976,-116.169,-35.809,179.375,5.301,149.109
C06165=1227.972,-115.919,-35.819,179.378,5.301,149.109
C06166=1227.966,-115.670,-35.829,179.380,5.301,149.108
C06167=1227.961,-115.420,-35.839,179.382,5.302,149.107
C06168=1227.956,-115.170,-35.848,179.384,5.301,149.107
C06169=1227.950,-114.920,-35.858,179.387,5.302,149.106
C06170=1227.945,-114.670,-35.869,179.389,5.301,149.105
C06171=1227.940,-114.420,-35.879,179.391,5.302,149.105
C06172=1227.935,-114.171,-35.889,179.394,5.301,149.104
C06173=1227.929,-113.922,-35.899,179.396,5.301,149.103
C06174=1227.924,-113.671,-35.910,179.398,5.301,149.102
C06175=1227.919,-113.422,-35.919,179.400,5.301,149.102
C06176=1227.914,-113.173,-35.929,179.403,5.302,149.101
C06177=1227.908,-112.922,-35.939,179.405,5.301,149.100
C06178=1227.903,-112.672,-35.950,179.407,5.302,149.100
C06179=1227.898,-112.423,-35.959,179.409,5.301,149.099
C06180=1227.893,-112.173,-35.970,179.412,5.302,149.098
C06181=1227.887,-111.923,-35.980,179.414,5.302,149.098
C06182=1227.882,-111.674,-35.990,179.417,5.302,149.097
C06183=1227.877,-111.423,-36.001,179.419,5.302,149.096
C06184=1227.872,-111.174,-36.010,179.421,5.302,149.096
C06185=1227.866,-110.925,-36.021,179.423,5.302,149.095
C06186=1227.861,-110.674,-36.031,179.425,5.302,149.094
C06187=1227.856,-110.425,-36.041,179.428,5.302,149.094
C06188=1227.851,-110.176,-36.051,179.430,5.302,149.093
C06189=1227.846,-109.925,-36.062,179.433,5.302,149.092
C06190=1227.840,-109.676,-36.072,179.435,5.302,149.091
C06191=1227.835,-109.426,-36.082,179.438,5.302,149.091
C06192=1227.830,-109.176,-36.093,179.440,5.302,149.090
C06193=1227.825,-108.927,-36.102,179.442,5.303,149.089
C06194=1227.820,-108.677,-36.113,179.444,5.302,149.089
C06195=1227.814,-108.427,-36.123,179.447,5.303,149.088
C06196=1227.809,-108.178,-36.133,179.449,5.302,149.087
C06197=1227.804,-107.927,-36.144,179.451,5.303,149.087
C06198=1227.798,-107.678,-36.154,179.454,5.302,149.086
C06199=1227.794,-107.428,-36.164,179.456,5.302,149.085
C06200=1227.788,-107.178,-36.174,179.458,5.302,149.084
C06201=1227.783,-106.929,-36.184,179.460,5.302,149.084
C06202=1227.778,-106.678,-36.195,179.463,5.303,149.083
C06203=1227.772,-106.430,-36.206,179.465,5.303,149.083
C06204=1227.767,-106.179,-36.216,179.467,5.303,149.082
C06205=1227.762,-105.930,-36.227,179.469,5.303,149.081
C06206=1227.757,-105.681,-36.236,179.472,5.303,149.080
C06207=1227.752,-105.430,-36.247,179.474,5.303,149.080
C06208=1227.746,-105.181,-36.257,179.477,5.303,149.079
C06209=1227.741,-104.930,-36.268,179.479,5.303,149.078
C06210=1227.736,-104.681,-36.278,179.482,5.303,149.078
C06211=1227.730,-104.431,-36.288,179.484,5.303,149.077
C06212=1227.725,-104.182,-36.299,179.486,5.303,149.076
C06213=1227.720,-103.932,-36.309,179.489,5.303,149.075
C06214=1227.715,-103.682,-36.320,179.491,5.304,149.075
C06215=1227.709,-103.432,-36.330,179.493,5.303,149.074
C06216=1227.704,-103.182,-36.341,179.495,5.303,149.074
C06217=1227.699,-102.933,-36.350,179.498,5.303,149.073
C06218=1227.695,-102.683,-36.362,179.500,5.303,149.072
C06219=1227.689,-102.434,-36.372,179.502,5.303,149.071
C06220=1227.684,-102.184,-36.383,179.504,5.303,149.071
C06221=1227.678,-101.934,-36.393,179.507,5.304,149.070
C06222=1227.673,-101.684,-36.403,179.509,5.303,149.069
C06223=1227.668,-101.435,-36.414,179.512,5.304,149.069
C06224=1227.662,-101.185,-36.424,179.514,5.303,149.068
C06225=1227.657,-100.914,-36.436,179.517,5.304,149.067
C06226=1227.652,-100.643,-36.448,179.519,5.303,149.066
C06227=1227.645,-100.372,-36.459,179.521,5.304,149.066
C06228=1227.640,-100.101,-36.470,179.524,5.304,149.065
C06229=1227.635,-99.851,-36.481,179.526,5.304,149.064
C06230=1227.630,-99.602,-36.491,179.529,5.304,149.064
C06231=1227.625,-99.351,-36.502,179.531,5.304,149.063
C06232=1227.619,-99.103,-36.513,179.534,5.304,149.062
C06233=1227.614,-98.852,-36.523,179.536,5.304,149.061
C06234=1227.609,-98.603,-36.534,179.538,5.304,149.061
C06235=1227.604,-98.353,-36.545,179.540,5.304,149.060
C06236=1227.598,-98.104,-36.555,179.543,5.304,149.059
C06237=1227.593,-97.853,-36.566,179.545,5.304,149.059
C06238=1227.588,-97.604,-36.576,179.547,5.304,149.058
C06239=1227.583,-97.354,-36.587,179.550,5.305,149.057
C06240=1227.578,-97.105,-36.597,179.552,5.304,149.057
C06241=1227.572,-96.854,-36.608,179.554,5.305,149.056
C06242=1227.567,-96.605,-36.619,179.556,5.304,149.055
C06243=1227.562,-96.355,-36.630,179.559,5.305,149.054
C06244=1227.556,-96.106,-36.641,179.561,5.304,149.054
C06245=1227.551,-95.856,-36.651,179.564,5.305,149.053
C06246=1227.546,-95.605,-36.662,179.566,5.304,149.052
C06247=1227.541,-95.357,-36.673,179.569,5.305,149.052
C06248=1227.536,-95.106,-36.684,179.571,5.305,149.051
C06249=1227.530,-94.857,-36.694,179.573,5.305,149.050
C06250=1227.526,-94.607,-36.705,179.575,5.305,149.050
C06251=1227.520,-94.358,-36.715,179.578,5.305,149.049
C06252=1227.515,-94.108,-36.727,179.580,5.305,149.048
C06253=1227.509,-93.858,-36.737,179.583,5.305,149.047
C06254=1227.504,-93.608,-36.749,179.584,5.305,149.047
C06255=1227.499,-93.358,-36.759,179.587,5.306,149.046
C06256=1227.494,-93.109,-36.769,179.589,5.305,149.045
C06257=1227.489,-92.859,-36.781,179.592,5.306,149.045
C06258=1227.483,-92.610,-36.791,179.594,5.305,149.044
C06259=1227.479,-92.360,-36.802,179.597,5.306,149.043
C06260=1227.473,-92.110,-36.812,179.599,5.305,149.043
C06261=1227.468,-91.860,-36.824,179.601,5.306,149.042
C06262=1227.463,-91.610,-36.835,179.604,5.306,149.041
C06263=1227.457,-91.361,-36.846,179.606,5.306,149.040
C06264=1227.452,-91.111,-36.856,179.608,5.306,149.040
C06265=1227.447,-90.862,-36.867,179.611,5.306,149.039
C06266=1227.442,-90.612,-36.878,179.613,5.306,149.038
C06267=1227.437,-90.362,-36.890,179.616,5.306,149.038
C06268=1227.431,-90.112,-36.900,179.618,5.306,149.037
C06269=1227.426,-89.863,-36.911,179.621,5.306,149.036
C06270=1227.421,-89.612,-36.922,179.623,5.306,149.035
C06271=1227.416,-89.364,-36.933,179.625,5.306,149.035
C06272=1227.411,-89.114,-36.945,179.627,5.306,149.034
C06273=1227.405,-88.864,-36.955,179.630,5.307,149.034
C06274=1227.400,-88.614,-36.966,179.632,5.306,149.033
C06275=1227.395,-88.364,-36.977,179.634,5.307,149.032
C06276=1227.390,-88.115,-36.988,179.636,5.307,149.031
C06277=1227.384,-87.865,-36.999,179.639,5.307,149.031
C06278=1227.380,-87.615,-37.010,179.641,5.307,149.030
C06279=1227.374,-87.366,-37.021,179.644,5.307,149.029
C06280=1227.369,-87.116,-37.032,179.646,5.307,149.029
C06281=1227.364,-86.866,-37.043,179.649,5.307,149.028
C06282=1227.359,-86.617,-37.054,179.651,5.307,149.027
C06283=1227.354,-86.367,-37.065,179.653,5.307,149.026
C06284=1227.349,-86.117,-37.076,179.655,5.307,149.026
C06285=1227.343,-85.867,-37.087,179.658,5.307,149.025
C06286=1227.338,-85.618,-37.098,179.660,5.307,149.024
C06287=1227.333,-85.368,-37.110,179.663,5.307,149.024
C06288=1227.328,-85.119,-37.120,179.665,5.307,149.023
C06289=1227.322,-84.869,-37.132,179.668,5.308,149.022
C06290=1227.318,-84.619,-37.143,179.670,5.307,149.022
C06291=1227.313,-84.369,-37.154,179.672,5.308,149.021
C06292=1227.307,-84.119,-37.165,179.675,5.307,149.020
C06293=1227.302,-83.870,-37.176,179.677,5.308,149.019
C06294=1227.297,-83.620,-37.188,179.679,5.307,149.019
C06295=1227.291,-83.370,-37.199,179.681,5.308,149.018
C06296=1227.286,-83.121,-37.210,179.684,5.308,149.017
C06297=1227.281,-82.871,-37.221,179.686,5.308,149.017
C06298=1227.276,-82.621,-37.233,179.688,5.308,149.016
C06299=1227.270,-82.372,-37.243,179.691,5.308,149.015
C06300=1227.266,-82.122,-37.254,179.693,5.308,149.015
C06301=1227.260,-81.872,-37.266,179.696,5.309,149.014
C06302=1227.255,-81.623,-37.277,179.698,5.308,149.013
C06303=1227.250,-81.373,-37.288,179.701,5.309,149.013
C06304=1227.245,-81.123,-37.300,179.703,5.308,149.012
C06305=1227.240,-80.873,-37.311,179.705,5.309,149.011
C06306=1227.235,-80.624,-37.322,179.707,5.308,149.010
C06307=1227.229,-80.374,-37.333,179.710,5.309,149.010
C06308=1227.224,-80.124,-37.344,179.712,5.309,149.009
C06309=1227.219,-79.874,-37.356,179.715,5.309,149.008
C06310=1227.213,-79.625,-37.367,179.717,5.309,149.008
C06311=1227.209,-79.376,-37.379,179.720,5.309,149.007
C06312=1227.203,-79.126,-37.390,179.722,5.309,149.006
C06313=1227.198,-78.876,-37.401,179.724,5.309,149.005
C06314=1227.193,-78.626,-37.413,179.726,5.309,149.005
C06315=1227.188,-78.377,-37.424,179.729,5.309,149.004
C06316=1227.183,-78.127,-37.435,179.731,5.309,149.003
C06317=1227.178,-77.877,-37.447,179.734,5.309,149.003
C06318=1227.173,-77.628,-37.458,179.736,5.309,149.002
C06319=1227.167,-77.378,-37.470,179.739,5.310,149.001
C06320=1227.162,-77.129,-37.481,179.741,5.310,149.000
C06321=1227.156,-76.878,-37.492,179.743,5.310,149.000
C06322=1227.152,-76.628,-37.504,179.746,5.310,148.999
C06323=1227.147,-76.379,-37.515,179.748,5.310,148.998
C06324=1227.141,-76.130,-37.526,179.751,5.310,148.998
C06325=1227.136,-75.880,-37.538,179.753,5.310,148.997
C06326=1227.131,-75.630,-37.549,179.756,5.310,148.996
C06327=1227.126,-75.380,-37.561,179.758,5.310,148.995
C06328=1227.121,-75.131,-37.573,179.760,5.310,148.995
C06329=1227.114,-74.860,-37.585,179.762,5.310,148.994
C06330=1227.109,-74.590,-37.598,179.765,5.311,148.993
C06331=1227.104,-74.319,-37.610,179.768,5.311,148.993
C06332=1227.098,-74.049,-37.622,179.770,5.311,148.992
C06333=1227.093,-73.800,-37.634,179.773,5.311,148.991
C06334=1227.088,-73.550,-37.646,179.775,5.311,148.991
C06335=1227.083,-73.300,-37.657,179.777,5.311,148.990
C06336=1227.077,-73.050,-37.669,179.779,5.311,148.989
C06337=1227.072,-72.801,-37.680,179.782,5.311,148.988
C06338=1227.067,-72.551,-37.692,179.784,5.311,148.988
C06339=1227.062,-72.302,-37.703,179.787,5.311,148.987
C06340=1227.057,-72.052,-37.715,179.789,5.312,148.986
C06341=1227.052,-71.802,-37.726,179.792,5.312,148.986
C06342=1227.046,-71.552,-37.738,179.794,5.312,148.985
C06343=1227.041,-71.302,-37.750,179.796,5.312,148.984
C06344=1227.036,-71.053,-37.761,179.799,5.312,148.983
C06345=1227.030,-70.803,-37.773,179.801,5.312,148.983
C06346=1227.026,-70.554,-37.784,179.804,5.312,148.982
C06347=1227.020,-70.304,-37.796,179.806,5.312,148.981
C06348=1227.016,-70.055,-37.808,179.808,5.312,148.981
C06349=1227.010,-69.805,-37.820,179.811,5.312,148.980
C06350=1227.005,-69.555,-37.832,179.813,5.312,148.979
C06351=1227.000,-69.305,-37.843,179.815,5.312,148.978
C06352=1226.994,-69.056,-37.854,179.818,5.313,148.978
C06353=1226.990,-68.806,-37.866,179.820,5.312,148.977
C06354=1226.984,-68.556,-37.878,179.823,5.313,148.976
C06355=1226.979,-68.307,-37.889,179.825,5.313,148.976
C06356=1226.974,-68.057,-37.901,179.828,5.313,148.975
C06357=1226.969,-67.808,-37.913,179.830,5.313,148.974
C06358=1226.963,-67.558,-37.925,179.832,5.313,148.974
C06359=1226.959,-67.308,-37.936,179.835,5.313,148.973
C06360=1226.953,-67.058,-37.948,179.837,5.313,148.972
C06361=1226.948,-66.808,-37.960,179.840,5.314,148.971
C06362=1226.943,-66.559,-37.972,179.842,5.313,148.971
C06363=1226.938,-66.309,-37.984,179.844,5.314,148.970
C06364=1226.933,-66.059,-37.996,179.847,5.313,148.969
C06365=1226.927,-65.810,-38.007,179.849,5.314,148.969
C06366=1226.922,-65.560,-38.019,179.852,5.314,148.968
C06367=1226.917,-65.311,-38.031,179.854,5.314,148.967
C06368=1226.912,-65.061,-38.043,179.857,5.314,148.966
C06369=1226.907,-64.812,-38.055,179.859,5.314,148.966
C06370=1226.901,-64.562,-38.066,179.861,5.315,148.965
C06371=1226.897,-64.313,-38.078,179.863,5.314,148.964
C06372=1226.891,-64.063,-38.090,179.866,5.315,148.964
C06373=1226.886,-63.813,-38.102,179.868,5.314,148.963
C06374=1226.881,-63.563,-38.114,179.871,5.315,148.962
C06375=1226.876,-63.314,-38.126,179.873,5.314,148.962
C06376=1226.871,-63.064,-38.138,179.876,5.315,148.961
C06377=1226.865,-62.814,-38.150,179.878,5.315,148.960
C06378=1226.861,-62.564,-38.161,179.880,5.315,148.959
C06379=1226.855,-62.315,-38.174,179.883,5.316,148.959
C06380=1226.850,-62.065,-38.186,179.885,5.315,148.958
C06381=1226.845,-61.815,-38.198,179.888,5.316,148.957
C06382=1226.840,-61.566,-38.210,179.890,5.315,148.957
C06383=1226.835,-61.316,-38.221,179.893,5.316,148.956
C06384=1226.829,-61.066,-38.233,179.895,5.315,148.955
C06385=1226.824,-60.817,-38.246,179.897,5.316,148.954
C06386=1226.820,-60.567,-38.257,179.900,5.316,148.954
C06387=1226.814,-60.318,-38.270,179.902,5.316,148.953
C06388=1226.809,-60.068,-38.282,179.905,5.317,148.952
C06389=1226.804,-59.818,-38.294,179.907,5.316,148.952
C06390=1226.798,-59.569,-38.306,179.910,5.317,148.951
C06391=1226.794,-59.319,-38.318,179.912,5.316,148.950
C06392=1226.788,-59.069,-38.329,179.914,5.317,148.950
C06393=1226.783,-58.820,-38.342,179.916,5.316,148.949
C06394=1226.778,-58.570,-38.354,179.919,5.317,148.948
C06395=1226.773,-58.321,-38.366,179.922,5.317,148.947
C06396=1226.768,-58.071,-38.378,179.924,5.317,148.947
C06397=1226.763,-57.821,-38.391,179.926,5.318,148.946
C06398=1226.758,-57.571,-38.403,179.929,5.317,148.945
C06399=1226.753,-57.321,-38.415,179.931,5.318,148.945
C06400=1226.747,-57.072,-38.427,179.933,5.317,148.944
C06401=1226.742,-56.822,-38.439,179.936,5.318,148.943
C06402=1226.737,-56.573,-38.452,179.939,5.318,148.942
C06403=1226.732,-56.323,-38.463,179.941,5.318,148.942
C06404=1226.727,-56.074,-38.475,179.943,5.318,148.941
C06405=1226.722,-55.824,-38.487,179.945,5.318,148.940
C06406=1226.717,-55.574,-38.500,179.948,5.319,148.940
C06407=1226.711,-55.324,-38.512,179.950,5.318,148.939
C06408=1226.706,-55.075,-38.524,179.953,5.319,148.938
C06409=1226.701,-54.824,-38.537,179.956,5.319,148.938
C06410=1226.696,-54.575,-38.549,179.958,5.319,148.937
C06411=1226.691,-54.326,-38.561,179.960,5.319,148.936
C06412=1226.686,-54.076,-38.573,179.962,5.319,148.935
C06413=1226.681,-53.827,-38.586,179.965,5.320,148.935
C06414=1226.676,-53.577,-38.598,179.967,5.319,148.934
C06415=1226.671,-53.328,-38.610,179.970,5.320,148.933
C06416=1226.665,-53.078,-38.622,179.973,5.320,148.933
C06417=1226.660,-52.828,-38.635,179.975,5.320,148.932
C06418=1226.655,-52.578,-38.647,179.977,5.320,148.931
C06419=1226.650,-52.328,-38.660,179.979,5.320,148.931
C06420=1226.645,-52.079,-38.672,179.982,5.320,148.930
C06421=1226.639,-51.829,-38.684,179.984,5.320,148.929
C06422=1226.634,-51.580,-38.697,179.987,5.321,148.928
C06423=1226.629,-51.330,-38.709,179.989,5.321,148.928
C06424=1226.624,-51.081,-38.721,179.992,5.321,148.927
C06425=1226.619,-50.831,-38.734,179.994,5.321,148.926
C06426=1226.614,-50.581,-38.746,179.996,5.321,148.926
C06427=1226.609,-50.331,-38.759,179.999,5.321,148.925
C06428=1226.604,-50.082,-38.771,-179.998,5.322,148.924
C06429=1226.598,-49.832,-38.783,-179.996,5.322,148.923
C06430=1226.593,-49.583,-38.796,-179.994,5.322,148.923
C06431=1226.589,-49.333,-38.809,-179.992,5.322,148.922
C06432=1226.583,-49.083,-38.821,-179.989,5.322,148.921
C06433=1226.577,-48.814,-38.834,-179.986,5.323,148.921
C06434=1226.572,-48.544,-38.848,-179.984,5.322,148.920
C06435=1226.567,-48.274,-38.861,-179.981,5.322,148.919
C06436=1226.561,-48.004,-38.874,-179.978,5.323,148.918
C06437=1226.556,-47.754,-38.887,-179.976,5.323,148.918
C06438=1226.551,-47.504,-38.899,-179.974,5.323,148.917
C06439=1226.546,-47.255,-38.912,-179.971,5.324,148.916
C06440=1226.541,-47.006,-38.925,-179.969,5.323,148.916
C06441=1226.536,-46.756,-38.937,-179.966,5.324,148.915
C06442=1226.531,-46.506,-38.949,-179.964,5.323,148.914
C06443=1226.526,-46.256,-38.962,-179.961,5.324,148.913
C06444=1226.520,-46.007,-38.975,-179.959,5.324,148.913
C06445=1226.515,-45.758,-38.987,-179.957,5.324,148.912
C06446=1226.510,-45.509,-39.000,-179.954,5.324,148.911
C06447=1226.505,-45.258,-39.013,-179.952,5.324,148.911
C06448=1226.500,-45.008,-39.025,-179.949,5.325,148.910
C06449=1226.494,-44.759,-39.038,-179.947,5.324,148.909
C06450=1226.489,-44.510,-39.050,-179.944,5.325,148.909
C06451=1226.485,-44.260,-39.063,-179.942,5.325,148.908
C06452=1226.479,-44.010,-39.075,-179.940,5.325,148.907
C06453=1226.474,-43.760,-39.088,-179.937,5.325,148.906
C06454=1226.469,-43.511,-39.100,-179.935,5.325,148.906
C06455=1226.464,-43.261,-39.114,-179.932,5.326,148.905
C06456=1226.459,-43.011,-39.127,-179.930,5.326,148.904
C06457=1226.454,-42.762,-39.139,-179.928,5.326,148.904
C06458=1226.448,-42.513,-39.152,-179.925,5.326,148.903
C06459=1226.444,-42.263,-39.165,-179.923,5.326,148.902
C06460=1226.438,-42.013,-39.177,-179.920,5.326,148.902
C06461=1226.433,-41.763,-39.189,-179.917,5.327,148.901
C06462=1226.427,-41.514,-39.202,-179.915,5.327,148.900
C06463=1226.423,-41.264,-39.215,-179.913,5.327,148.899
C06464=1226.418,-41.015,-39.228,-179.910,5.328,148.899
C06465=1226.413,-40.765,-39.241,-179.908,5.327,148.898
C06466=1226.408,-40.515,-39.254,-179.905,5.328,148.897
C06467=1226.402,-40.266,-39.267,-179.903,5.327,148.897
C06468=1226.397,-40.016,-39.279,-179.900,5.327,148.896
C06469=1226.392,-39.767,-39.292,-179.897,5.328,148.895
C06470=1226.388,-39.517,-39.305,-179.895,5.328,148.894
C06471=1226.382,-39.268,-39.318,-179.893,5.328,148.894
C06472=1226.377,-39.018,-39.331,-179.891,5.328,148.893
C06473=1226.372,-38.768,-39.344,-179.888,5.328,148.892
C06474=1226.367,-38.519,-39.356,-179.885,5.329,148.891
C06475=1226.362,-38.269,-39.369,-179.883,5.328,148.891
C06476=1226.357,-38.019,-39.383,-179.881,5.329,148.890
C06477=1226.351,-37.770,-39.395,-179.878,5.329,148.889
C06478=1226.346,-37.520,-39.408,-179.876,5.329,148.889
C06479=1226.342,-37.270,-39.421,-179.873,5.330,148.888
C06480=1226.336,-37.021,-39.434,-179.871,5.329,148.887
C06481=1226.331,-36.771,-39.446,-179.868,5.330,148.887
C06482=1226.326,-36.521,-39.459,-179.866,5.330,148.886
C06483=1226.320,-36.272,-39.473,-179.864,5.330,148.885
C06484=1226.315,-36.022,-39.485,-179.861,5.330,148.884
C06485=1226.311,-35.772,-39.498,-179.859,5.330,148.884
C06486=1226.306,-35.523,-39.511,-179.856,5.331,148.883
C06487=1226.300,-35.273,-39.524,-179.854,5.331,148.882
C06488=1226.295,-35.023,-39.537,-179.851,5.331,148.882
C06489=1226.290,-34.775,-39.550,-179.849,5.331,148.881
C06490=1226.285,-34.524,-39.564,-179.846,5.332,148.880
C06491=1226.280,-34.275,-39.576,-179.844,5.331,148.880
C06492=1226.275,-34.026,-39.589,-179.841,5.332,148.879
C06493=1226.270,-33.775,-39.603,-179.839,5.332,148.878
C06494=1226.265,-33.526,-39.615,-179.837,5.332,148.877
C06495=1226.259,-33.277,-39.628,-179.834,5.333,148.877
C06496=1226.254,-33.026,-39.641,-179.832,5.332,148.876
C06497=1226.249,-32.778,-39.655,-179.829,5.333,148.875
C06498=1226.245,-32.528,-39.668,-179.827,5.333,148.875
C06499=1226.239,-32.278,-39.681,-179.825,5.333,148.874
C06500=1226.234,-32.029,-39.693,-179.822,5.334,148.873
C06501=1226.229,-31.778,-39.707,-179.819,5.334,148.873
C06502=1226.224,-31.530,-39.720,-179.817,5.334,148.872
C06503=1226.219,-31.280,-39.733,-179.814,5.334,148.871
C06504=1226.213,-31.030,-39.746,-179.812,5.334,148.870
C06505=1226.209,-30.780,-39.759,-179.810,5.334,148.870
C06506=1226.203,-30.530,-39.773,-179.807,5.335,148.869
C06507=1226.198,-30.282,-39.786,-179.805,5.335,148.868
C06508=1226.194,-30.032,-39.799,-179.802,5.335,148.868
C06509=1226.188,-29.782,-39.812,-179.800,5.336,148.867
C06510=1226.183,-29.532,-39.825,-179.798,5.335,148.866
C06511=1226.178,-29.283,-39.839,-179.795,5.336,148.866
C06512=1226.173,-29.033,-39.852,-179.792,5.336,148.865
C06513=1226.168,-28.784,-39.865,-179.790,5.336,148.864
C06514=1226.163,-28.534,-39.879,-179.787,5.336,148.864
C06515=1226.158,-28.285,-39.891,-179.785,5.337,148.863
C06516=1226.152,-28.035,-39.905,-179.783,5.337,148.862
C06517=1226.148,-27.785,-39.918,-179.780,5.337,148.861
C06518=1226.142,-27.536,-39.932,-179.778,5.337,148.861
C06519=1226.138,-27.286,-39.944,-179.775,5.337,148.860
C06520=1226.132,-27.036,-39.958,-179.773,5.338,148.859
C06521=1226.127,-26.787,-39.971,-179.771,5.337,148.859
C06522=1226.122,-26.537,-39.985,-179.768,5.338,148.858
C06523=1226.117,-26.288,-39.998,-179.765,5.338,148.857
C06524=1226.111,-26.038,-40.011,-179.763,5.338,148.857
C06525=1226.107,-25.788,-40.024,-179.761,5.339,148.856
C06526=1226.101,-25.539,-40.038,-179.758,5.339,148.855
C06527=1226.097,-25.289,-40.051,-179.756,5.339,148.854
C06528=1226.091,-25.040,-40.064,-179.753,5.339,148.854
C06529=1226.087,-24.790,-40.078,-179.750,5.340,148.853
C06530=1226.081,-24.541,-40.091,-179.748,5.340,148.852
C06531=1226.077,-24.291,-40.105,-179.746,5.340,148.852
C06532=1226.071,-24.042,-40.118,-179.743,5.341,148.851
C06533=1226.067,-23.792,-40.132,-179.741,5.340,148.850
C06534=1226.061,-23.542,-40.145,-179.738,5.341,148.850
C06535=1226.056,-23.293,-40.158,-179.736,5.341,148.849
C06536=1226.051,-23.043,-40.172,-179.734,5.341,148.848
C06537=1226.045,-22.774,-40.187,-179.730,5.341,148.847
C06538=1226.040,-22.504,-40.201,-179.728,5.342,148.847
C06539=1226.035,-22.235,-40.216,-179.725,5.342,148.846
C06540=1226.029,-21.966,-40.231,-179.723,5.342,148.845
C06541=1226.024,-21.716,-40.244,-179.720,5.342,148.844
C06542=1226.019,-21.467,-40.258,-179.718,5.343,148.844
C06543=1226.013,-21.217,-40.271,-179.716,5.342,148.843
C06544=1226.009,-20.968,-40.284,-179.713,5.343,148.842
C06545=1226.003,-20.718,-40.298,-179.710,5.343,148.842
C06546=1225.998,-20.468,-40.312,-179.708,5.343,148.841
C06547=1225.993,-20.219,-40.324,-179.706,5.344,148.840
C06548=1225.988,-19.969,-40.339,-179.703,5.344,148.840
C06549=1225.983,-19.719,-40.353,-179.701,5.344,148.839
C06550=1225.978,-19.470,-40.366,-179.698,5.344,148.838
C06551=1225.973,-19.220,-40.380,-179.696,5.345,148.838
C06552=1225.968,-18.971,-40.393,-179.693,5.345,148.837
C06553=1225.963,-18.721,-40.407,-179.691,5.345,148.836
C06554=1225.958,-18.471,-40.420,-179.688,5.346,148.835
C06555=1225.953,-18.222,-40.434,-179.685,5.346,148.835
C06556=1225.948,-17.973,-40.448,-179.683,5.346,148.834
C06557=1225.942,-17.723,-40.461,-179.681,5.346,148.833
C06558=1225.937,-17.473,-40.475,-179.678,5.347,148.833
C06559=1225.933,-17.224,-40.489,-179.676,5.346,148.832
C06560=1225.927,-16.974,-40.502,-179.673,5.347,148.831
C06561=1225.922,-16.725,-40.517,-179.671,5.347,148.831
C06562=1225.917,-16.475,-40.529,-179.669,5.347,148.830
C06563=1225.912,-16.226,-40.543,-179.666,5.348,148.829
C06564=1225.907,-15.976,-40.558,-179.663,5.348,148.828
C06565=1225.902,-15.727,-40.570,-179.661,5.348,148.828
C06566=1225.897,-15.477,-40.585,-179.659,5.348,148.827
C06567=1225.892,-15.227,-40.599,-179.656,5.349,148.826
C06568=1225.887,-14.978,-40.613,-179.654,5.349,148.826
C06569=1225.882,-14.728,-40.626,-179.651,5.349,148.825
C06570=1225.877,-14.478,-40.640,-179.648,5.350,148.824
C06571=1225.872,-14.229,-40.654,-179.646,5.350,148.824
C06572=1225.866,-13.979,-40.668,-179.644,5.350,148.823
C06573=1225.862,-13.730,-40.681,-179.641,5.350,148.822
C06574=1225.857,-13.481,-40.695,-179.638,5.351,148.822
C06575=1225.852,-13.231,-40.709,-179.636,5.351,148.821
C06576=1225.846,-12.981,-40.723,-179.634,5.351,148.820
C06577=1225.841,-12.732,-40.737,-179.631,5.352,148.819
C06578=1225.837,-12.482,-40.751,-179.629,5.351,148.819
C06579=1225.832,-12.232,-40.765,-179.626,5.352,148.818
C06580=1225.826,-11.983,-40.779,-179.624,5.352,148.817
C06581=1225.821,-11.733,-40.792,-179.622,5.352,148.817
C06582=1225.816,-11.483,-40.807,-179.619,5.353,148.816
C06583=1225.812,-11.234,-40.820,-179.616,5.353,148.815
C06584=1225.806,-10.985,-40.834,-179.614,5.354,148.815
C06585=1225.801,-10.735,-40.848,-179.612,5.353,148.814
C06586=1225.796,-10.485,-40.862,-179.609,5.354,148.813
C06587=1225.790,-10.236,-40.876,-179.606,5.354,148.813
C06588=1225.785,-9.986,-40.890,-179.604,5.354,148.812
C06589=1225.781,-9.737,-40.904,-179.601,5.354,148.811
C06590=1225.776,-9.487,-40.918,-179.599,5.355,148.810
C06591=1225.771,-9.238,-40.932,-179.596,5.356,148.810
C06592=1225.766,-8.988,-40.946,-179.594,5.355,148.809
C06593=1225.761,-8.739,-40.961,-179.591,5.356,148.808
C06594=1225.755,-8.489,-40.974,-179.589,5.356,148.808
C06595=1225.750,-8.239,-40.988,-179.587,5.356,148.807
C06596=1225.746,-7.990,-41.002,-179.584,5.356,148.806
C06597=1225.741,-7.740,-41.016,-179.581,5.357,148.806
C06598=1225.736,-7.491,-41.030,-179.579,5.357,148.805
C06599=1225.730,-7.242,-41.044,-179.577,5.357,148.804
C06600=1225.725,-6.992,-41.059,-179.574,5.358,148.804
C06601=1225.720,-6.742,-41.073,-179.571,5.358,148.803
C06602=1225.715,-6.492,-41.087,-179.569,5.358,148.802
C06603=1225.710,-6.243,-41.101,-179.567,5.358,148.801
C06604=1225.705,-5.994,-41.115,-179.564,5.359,148.801
C06605=1225.700,-5.744,-41.130,-179.561,5.359,148.800
C06606=1225.695,-5.494,-41.144,-179.559,5.359,148.799
C06607=1225.690,-5.245,-41.158,-179.557,5.360,148.799
C06608=1225.685,-4.996,-41.171,-179.554,5.360,148.798
C06609=1225.680,-4.746,-41.186,-179.552,5.360,148.797
C06610=1225.675,-4.496,-41.200,-179.549,5.360,148.797
C06611=1225.670,-4.247,-41.214,-179.547,5.361,148.796
C06612=1225.665,-3.997,-41.229,-179.544,5.361,148.795
C06613=1225.660,-3.748,-41.242,-179.542,5.361,148.795
C06614=1225.655,-3.498,-41.257,-179.539,5.362,148.794
C06615=1225.650,-3.249,-41.271,-179.536,5.362,148.793
C06616=1225.645,-2.999,-41.285,-179.534,5.363,148.793
C06617=1225.640,-2.749,-41.300,-179.532,5.362,148.792
C06618=1225.635,-2.500,-41.313,-179.529,5.363,148.791
C06619=1225.630,-2.250,-41.328,-179.526,5.363,148.790
C06620=1225.625,-2.001,-41.343,-179.524,5.363,148.790
C06621=1225.620,-1.752,-41.357,-179.522,5.364,148.789
C06622=1225.615,-1.502,-41.371,-179.519,5.364,148.788
C06623=1225.610,-1.252,-41.386,-179.516,5.365,148.788
C06624=1225.605,-1.003,-41.399,-179.514,5.364,148.787
C06625=1225.599,-0.753,-41.414,-179.512,5.365,148.786
C06626=1225.594,-0.503,-41.429,-179.509,5.365,148.786
C06627=1225.589,-0.254,-41.443,-179.506,5.366,148.785
C06628=1225.584,-0.005,-41.458,-179.504,5.366,148.784
C06629=1225.579,0.245,-41.472,-179.502,5.366,148.784
C06630=1225.574,0.495,-41.486,-179.499,5.367,148.783
C06631=1225.569,0.744,-41.500,-179.496,5.367,148.782
C06632=1225.564,0.993,-41.515,-179.494,5.367,148.781
C06633=1225.559,1.243,-41.529,-179.492,5.368,148.781
C06634=1225.554,1.492,-41.544,-179.489,5.368,148.780
C06635=1225.549,1.742,-41.558,-179.486,5.369,148.779
C06636=1225.544,1.992,-41.572,-179.484,5.368,148.779
C06637=1225.539,2.242,-41.587,-179.482,5.369,148.778
C06638=1225.534,2.491,-41.602,-179.479,5.369,148.777
C06639=1225.529,2.741,-41.617,-179.476,5.370,148.777
C06640=1225.524,2.990,-41.631,-179.474,5.370,148.776
C06641=1225.518,3.258,-41.646,-179.472,5.370,148.775
C06642=1225.513,3.527,-41.662,-179.469,5.371,148.775
C06643=1225.507,3.797,-41.677,-179.466,5.371,148.774
C06644=1225.502,4.066,-41.693,-179.463,5.371,148.773
C06645=1225.497,4.315,-41.708,-179.460,5.372,148.772
C06646=1225.492,4.564,-41.722,-179.458,5.372,148.772
C06647=1225.487,4.814,-41.737,-179.456,5.372,148.771
C06648=1225.482,5.064,-41.751,-179.453,5.373,148.770
C06649=1225.477,5.313,-41.767,-179.450,5.373,148.770
C06650=1225.472,5.563,-41.781,-179.448,5.373,148.769
C06651=1225.467,5.813,-41.795,-179.446,5.373,148.768
C06652=1225.462,6.062,-41.810,-179.443,5.374,148.767
C06653=1225.457,6.311,-41.824,-179.441,5.375,148.767
C06654=1225.452,6.561,-41.840,-179.438,5.375,148.766
C06655=1225.447,6.811,-41.854,-179.436,5.375,148.766
C06656=1225.442,7.060,-41.868,-179.433,5.376,148.765
C06657=1225.437,7.309,-41.883,-179.431,5.376,148.764
C06658=1225.431,7.559,-41.898,-179.428,5.377,148.764
C06659=1225.427,7.808,-41.913,-179.426,5.376,148.763
C06660=1225.422,8.057,-41.927,-179.423,5.377,148.762
C06661=1225.417,8.307,-41.942,-179.421,5.377,148.762
C06662=1225.412,8.556,-41.957,-179.418,5.378,148.761
C06663=1225.406,8.806,-41.971,-179.416,5.378,148.760
C06664=1225.402,9.055,-41.986,-179.413,5.378,148.759
C06665=1225.397,9.305,-42.001,-179.411,5.379,148.759
C06666=1225.391,9.555,-42.016,-179.408,5.379,148.758
C06667=1225.386,9.804,-42.031,-179.405,5.380,148.757
C06668=1225.381,10.054,-42.045,-179.403,5.379,148.757
C06669=1225.377,10.303,-42.060,-179.401,5.380,148.756
C06670=1225.371,10.553,-42.075,-179.398,5.381,148.755
C06671=1225.366,10.802,-42.090,-179.395,5.381,148.755
C06672=1225.362,11.052,-42.104,-179.393,5.381,148.754
C06673=1225.356,11.301,-42.120,-179.391,5.381,148.753
C06674=1225.352,11.551,-42.135,-179.388,5.382,148.753
C06675=1225.347,11.801,-42.149,-179.385,5.382,148.752
C06676=1225.342,12.050,-42.165,-179.383,5.383,148.751
C06677=1225.337,12.300,-42.179,-179.381,5.383,148.751
C06678=1225.332,12.549,-42.194,-179.378,5.383,148.750
C06679=1225.326,12.799,-42.209,-179.375,5.384,148.749
C06680=1225.322,13.048,-42.224,-179.373,5.384,148.749
C06681=1225.317,13.298,-42.238,-179.370,5.385,148.748
C06682=1225.311,13.547,-42.254,-179.368,5.384,148.747
C06683=1225.307,13.796,-42.269,-179.365,5.385,148.746
C06684=1225.302,14.046,-42.283,-179.363,5.386,148.746
C06685=1225.296,14.295,-42.299,-179.361,5.386,148.745
C06686=1225.292,14.545,-42.313,-179.358,5.387,148.745
C06687=1225.286,14.795,-42.329,-179.356,5.387,148.744
C06688=1225.281,15.044,-42.344,-179.353,5.387,148.743
C06689=1225.277,15.293,-42.358,-179.351,5.388,148.743
C06690=1225.271,15.543,-42.373,-179.348,5.388,148.742
C06691=1225.267,15.793,-42.389,-179.345,5.389,148.741
C06692=1225.261,16.043,-42.404,-179.343,5.389,148.741
C06693=1225.257,16.292,-42.419,-179.341,5.389,148.740
C06694=1225.251,16.541,-42.434,-179.338,5.390,148.739
C06695=1225.246,16.791,-42.449,-179.335,5.390,148.738
C06696=1225.242,17.040,-42.464,-179.333,5.391,148.738
C06697=1225.236,17.289,-42.479,-179.331,5.390,148.737
C06698=1225.231,17.539,-42.493,-179.328,5.391,148.736
C06699=1225.226,17.788,-42.509,-179.325,5.391,148.736
C06700=1225.222,18.038,-42.524,-179.323,5.392,148.735
C06701=1225.217,18.288,-42.540,-179.320,5.393,148.734
C06702=1225.212,18.537,-42.554,-179.318,5.392,148.734
C06703=1225.206,18.787,-42.570,-179.315,5.393,148.733
C06704=1225.202,19.036,-42.585,-179.313,5.393,148.732
C06705=1225.196,19.285,-42.600,-179.310,5.394,148.732
C06706=1225.191,19.535,-42.615,-179.308,5.395,148.731
C06707=1225.186,19.785,-42.631,-179.305,5.395,148.731
C06708=1225.182,20.034,-42.646,-179.303,5.395,148.730
C06709=1225.176,20.283,-42.661,-179.300,5.396,148.729
C06710=1225.172,20.533,-42.676,-179.298,5.396,148.728
C06711=1225.166,20.783,-42.691,-179.295,5.397,148.728
C06712=1225.161,21.032,-42.706,-179.292,5.397,148.727
C06713=1225.157,21.282,-42.722,-179.290,5.397,148.726
C06714=1225.152,21.531,-42.737,-179.288,5.397,148.726
C06715=1225.147,21.780,-42.753,-179.285,5.398,148.725
C06716=1225.142,22.029,-42.768,-179.282,5.399,148.724
C06717=1225.136,22.279,-42.782,-179.280,5.399,148.724
C06718=1225.131,22.529,-42.798,-179.277,5.400,148.723
C06719=1225.127,22.779,-42.813,-179.275,5.399,148.722
C06720=1225.121,23.028,-42.829,-179.272,5.400,148.722
C06721=1225.117,23.277,-42.844,-179.270,5.400,148.721
C06722=1225.111,23.526,-42.860,-179.267,5.401,148.720
C06723=1225.107,23.776,-42.875,-179.265,5.402,148.720
C06724=1225.102,24.026,-42.890,-179.262,5.402,148.719
C06725=1225.097,24.275,-42.906,-179.260,5.402,148.718
C06726=1225.092,24.524,-42.921,-179.258,5.403,148.718
C06727=1225.087,24.774,-42.937,-179.255,5.403,148.717
C06728=1225.083,25.023,-42.952,-179.252,5.404,148.716
C06729=1225.077,25.273,-42.967,-179.250,5.404,148.716
C06730=1225.071,25.523,-42.982,-179.247,5.405,148.715
C06731=1225.067,25.772,-42.997,-179.245,5.405,148.714
C06732=1225.062,26.022,-43.013,-179.242,5.405,148.714
C06733=1225.057,26.271,-43.029,-179.240,5.406,148.713
C06734=1225.052,26.520,-43.044,-179.237,5.406,148.712
C06735=1225.047,26.770,-43.060,-179.234,5.407,148.712
C06736=1225.042,27.020,-43.076,-179.232,5.407,148.711
C06737=1225.037,27.269,-43.091,-179.229,5.408,148.710
C06738=1225.032,27.518,-43.106,-179.228,5.408,148.710
C06739=1225.027,27.767,-43.122,-179.225,5.408,148.709
C06740=1225.023,28.017,-43.138,-179.222,5.409,148.709
C06741=1225.017,28.266,-43.153,-179.220,5.410,148.708
C06742=1225.012,28.516,-43.169,-179.217,5.410,148.707
C06743=1225.007,28.765,-43.184,-179.214,5.411,148.706
C06744=1225.002,29.015,-43.200,-179.212,5.411,148.706
C06745=1224.997,29.284,-43.217,-179.209,5.412,148.705
C06746=1224.991,29.553,-43.233,-179.206,5.412,148.704
C06747=1224.985,29.821,-43.250,-179.204,5.413,148.704
C06748=1224.981,30.089,-43.267,-179.201,5.413,148.703
C06749=1224.976,30.339,-43.283,-179.199,5.413,148.702
C06750=1224.970,30.589,-43.298,-179.196,5.414,148.702
C06751=1224.965,30.838,-43.315,-179.194,5.414,148.701
C06752=1224.961,31.087,-43.330,-179.191,5.415,148.700
C06753=1224.956,31.337,-43.345,-179.188,5.415,148.700
C06754=1224.951,31.586,-43.361,-179.186,5.416,148.699
C06755=1224.946,31.836,-43.377,-179.183,5.416,148.698
C06756=1224.941,32.085,-43.392,-179.181,5.416,148.698
C06757=1224.936,32.334,-43.408,-179.178,5.417,148.697
C06758=1224.931,32.584,-43.424,-179.176,5.417,148.696
C06759=1224.926,32.834,-43.440,-179.173,5.418,148.696
C06760=1224.920,33.083,-43.455,-179.171,5.418,148.695
C06761=1224.916,33.333,-43.471,-179.168,5.419,148.694
C06762=1224.911,33.582,-43.487,-179.166,5.420,148.694
C06763=1224.906,33.831,-43.503,-179.163,5.420,148.693
C06764=1224.901,34.081,-43.519,-179.161,5.420,148.692
C06765=1224.896,34.331,-43.534,-179.158,5.421,148.692
C06766=1224.891,34.580,-43.551,-179.156,5.421,148.691
C06767=1224.887,34.829,-43.566,-179.153,5.422,148.690
C06768=1224.881,35.078,-43.581,-179.150,5.422,148.690
C06769=1224.876,35.329,-43.597,-179.148,5.423,148.689
C06770=1224.871,35.577,-43.614,-179.145,5.423,148.688
C06771=1224.866,35.827,-43.629,-179.143,5.424,148.688
C06772=1224.861,36.077,-43.645,-179.140,5.425,148.687
C06773=1224.856,36.326,-43.662,-179.138,5.425,148.687
C06774=1224.852,36.575,-43.677,-179.136,5.425,148.686
C06775=1224.847,36.825,-43.693,-179.133,5.426,148.685
C06776=1224.842,37.074,-43.709,-179.130,5.426,148.685
C06777=1224.837,37.324,-43.725,-179.128,5.427,148.684
C06778=1224.831,37.573,-43.740,-179.125,5.427,148.683
C06779=1224.827,37.823,-43.757,-179.122,5.428,148.683
C06780=1224.822,38.072,-43.773,-179.120,5.428,148.682
C06781=1224.817,38.321,-43.789,-179.117,5.429,148.681
C06782=1224.812,38.571,-43.805,-179.115,5.429,148.681
C06783=1224.806,38.820,-43.820,-179.113,5.430,148.680
C06784=1224.802,39.070,-43.837,-179.110,5.430,148.679
C06785=1224.796,39.319,-43.853,-179.108,5.431,148.679
C06786=1224.792,39.569,-43.869,-179.105,5.431,148.678
C06787=1224.787,39.818,-43.885,-179.102,5.432,148.677
C06788=1224.782,40.068,-43.901,-179.100,5.432,148.677
C06789=1224.777,40.317,-43.917,-179.097,5.433,148.676
C06790=1224.772,40.566,-43.932,-179.094,5.434,148.675
C06791=1224.768,40.816,-43.949,-179.092,5.434,148.675
C06792=1224.762,41.065,-43.964,-179.090,5.434,148.674
C06793=1224.758,41.314,-43.981,-179.088,5.435,148.674
C06794=1224.752,41.564,-43.997,-179.085,5.435,148.673
C06795=1224.748,41.813,-44.013,-179.082,5.436,148.672
C06796=1224.742,42.063,-44.029,-179.080,5.436,148.672
C06797=1224.737,42.313,-44.046,-179.077,5.437,148.671
C06798=1224.732,42.562,-44.062,-179.074,5.438,148.670
C06799=1224.727,42.811,-44.079,-179.072,5.438,148.670
C06800=1224.722,43.061,-44.094,-179.069,5.439,148.669
C06801=1224.718,43.310,-44.111,-179.067,5.440,148.668
C06802=1224.712,43.559,-44.127,-179.064,5.440,148.668
C06803=1224.708,43.809,-44.143,-179.062,5.441,148.667
C06804=1224.703,44.058,-44.159,-179.060,5.440,148.666
C06805=1224.698,44.308,-44.175,-179.057,5.441,148.666
C06806=1224.693,44.557,-44.192,-179.054,5.442,148.665
C06807=1224.688,44.807,-44.208,-179.052,5.442,148.664
C06808=1224.683,45.056,-44.224,-179.049,5.443,148.664
C06809=1224.678,45.305,-44.241,-179.047,5.444,148.663
C06810=1224.673,45.555,-44.256,-179.044,5.444,148.663
C06811=1224.669,45.804,-44.273,-179.042,5.445,148.662
C06812=1224.664,46.054,-44.289,-179.039,5.445,148.661
C06813=1224.658,46.303,-44.306,-179.036,5.446,148.661
C06814=1224.653,46.553,-44.322,-179.034,5.446,148.660
C06815=1224.648,46.802,-44.339,-179.031,5.447,148.659
C06816=1224.644,47.052,-44.355,-179.028,5.448,148.659
C06817=1224.638,47.300,-44.371,-179.026,5.448,148.658
C06818=1224.634,47.550,-44.388,-179.024,5.448,148.657
C06819=1224.629,47.799,-44.403,-179.022,5.449,148.657
C06820=1224.623,48.049,-44.420,-179.019,5.449,148.656
C06821=1224.619,48.299,-44.437,-179.016,5.450,148.655
C06822=1224.614,48.548,-44.453,-179.014,5.450,148.655
C06823=1224.609,48.798,-44.469,-179.011,5.451,148.654
C06824=1224.604,49.046,-44.486,-179.008,5.452,148.653
C06825=1224.599,49.296,-44.502,-179.006,5.453,148.653
C06826=1224.594,49.546,-44.519,-179.004,5.453,148.652
C06827=1224.589,49.795,-44.535,-179.001,5.454,148.652
C06828=1224.584,50.044,-44.552,-178.998,5.454,148.651
C06829=1224.579,50.293,-44.568,-178.996,5.455,148.650
C06830=1224.575,50.543,-44.585,-178.993,5.455,148.650
C06831=1224.569,50.793,-44.601,-178.990,5.456,148.649
C06832=1224.564,51.042,-44.618,-178.988,5.457,148.649
C06833=1224.560,51.291,-44.634,-178.986,5.457,148.648
C06834=1224.555,51.540,-44.651,-178.983,5.458,148.647
C06835=1224.550,51.790,-44.667,-178.980,5.459,148.647
C06836=1224.545,52.040,-44.684,-178.978,5.459,148.646
C06837=1224.540,52.289,-44.700,-178.975,5.460,148.645
C06838=1224.535,52.538,-44.717,-178.973,5.459,148.645
C06839=1224.531,52.788,-44.733,-178.971,5.460,148.644
C06840=1224.525,53.037,-44.750,-178.968,5.461,148.643
C06841=1224.520,53.286,-44.767,-178.966,5.461,148.643
C06842=1224.516,53.536,-44.784,-178.963,5.462,148.642
C06843=1224.510,53.785,-44.801,-178.960,5.463,148.641
C06844=1224.506,54.034,-44.817,-178.958,5.463,148.641
C06845=1224.501,54.285,-44.833,-178.956,5.464,148.640
C06846=1224.496,54.533,-44.850,-178.953,5.465,148.640
C06847=1224.490,54.783,-44.867,-178.950,5.465,148.639
C06848=1224.486,55.033,-44.883,-178.948,5.466,148.638
C06849=1224.481,55.301,-44.901,-178.945,5.466,148.638
C06850=1224.475,55.569,-44.920,-178.942,5.467,148.637
C06851=1224.470,55.837,-44.938,-178.939,5.468,148.636
C06852=1224.464,56.107,-44.956,-178.937,5.469,148.636
C06853=1224.459,56.356,-44.972,-178.934,5.469,148.635
C06854=1224.455,56.605,-44.989,-178.931,5.470,148.634
C06855=1224.450,56.855,-45.006,-178.929,5.471,148.634
C06856=1224.445,57.104,-45.022,-178.926,5.471,148.633
C06857=1224.440,57.353,-45.039,-178.924,5.472,148.633
C06858=1224.435,57.602,-45.057,-178.921,5.473,148.632
C06859=1224.431,57.852,-45.073,-178.919,5.473,148.631
C06860=1224.425,58.101,-45.090,-178.916,5.474,148.631
C06861=1224.420,58.350,-45.107,-178.913,5.474,148.630
C06862=1224.416,58.600,-45.124,-178.911,5.475,148.629
C06863=1224.411,58.850,-45.141,-178.909,5.475,148.629
C06864=1224.406,59.098,-45.157,-178.907,5.476,148.628
C06865=1224.400,59.348,-45.175,-178.904,5.476,148.627
C06866=1224.396,59.598,-45.191,-178.901,5.477,148.627
C06867=1224.390,59.847,-45.208,-178.899,5.477,148.626
C06868=1224.386,60.096,-45.225,-178.896,5.478,148.625
C06869=1224.381,60.346,-45.241,-178.894,5.479,148.625
C06870=1224.376,60.595,-45.259,-178.891,5.479,148.624
C06871=1224.372,60.844,-45.276,-178.889,5.480,148.624
C06872=1224.366,61.093,-45.293,-178.886,5.481,148.623
C06873=1224.361,61.343,-45.310,-178.883,5.481,148.622
C06874=1224.356,61.593,-45.327,-178.881,5.482,148.622
C06875=1224.352,61.842,-45.344,-178.879,5.483,148.621
C06876=1224.346,62.091,-45.360,-178.876,5.483,148.621
C06877=1224.342,62.340,-45.378,-178.873,5.484,148.620
C06878=1224.337,62.590,-45.395,-178.870,5.485,148.619
C06879=1224.332,62.839,-45.412,-178.867,5.486,148.619
C06880=1224.327,63.089,-45.429,-178.865,5.487,148.618
C06881=1224.322,63.337,-45.446,-178.863,5.487,148.617
C06882=1224.317,63.587,-45.463,-178.860,5.488,148.617
C06883=1224.312,63.837,-45.480,-178.857,5.488,148.616
C06884=1224.307,64.086,-45.497,-178.855,5.489,148.615
C06885=1224.303,64.335,-45.515,-178.853,5.490,148.615
C06886=1224.298,64.585,-45.532,-178.850,5.490,148.614
C06887=1224.293,64.834,-45.548,-178.847,5.491,148.614
C06888=1224.287,65.084,-45.565,-178.845,5.492,148.613
C06889=1224.283,65.333,-45.583,-178.842,5.492,148.612
C06890=1224.278,65.582,-45.600,-178.840,5.493,148.612
C06891=1224.273,65.832,-45.617,-178.837,5.494,148.611
C06892=1224.269,66.081,-45.635,-178.835,5.494,148.611
C06893=1224.263,66.330,-45.652,-178.832,5.495,148.610
C06894=1224.258,66.580,-45.668,-178.829,5.495,148.609
C06895=1224.253,66.829,-45.686,-178.827,5.496,148.609
C06896=1224.248,67.079,-45.704,-178.825,5.497,148.608
C06897=1224.244,67.328,-45.720,-178.822,5.498,148.608
C06898=1224.239,67.577,-45.738,-178.819,5.498,148.607
C06899=1224.234,67.827,-45.755,-178.817,5.499,148.606
C06900=1224.229,68.077,-45.772,-178.814,5.499,148.606
C06901=1224.224,68.325,-45.790,-178.812,5.500,148.605
C06902=1224.219,68.574,-45.806,-178.809,5.501,148.604
C06903=1224.214,68.824,-45.824,-178.807,5.501,148.604
C06904=1224.209,69.073,-45.842,-178.804,5.502,148.603
C06905=1224.205,69.322,-45.859,-178.802,5.503,148.603
C06906=1224.200,69.572,-45.876,-178.799,5.503,148.602
C06907=1224.195,69.822,-45.893,-178.797,5.504,148.601
C06908=1224.190,70.071,-45.911,-178.794,5.505,148.601
C06909=1224.185,70.321,-45.928,-178.792,5.505,148.600
C06910=1224.180,70.570,-45.946,-178.789,5.506,148.600
C06911=1224.176,70.819,-45.963,-178.787,5.507,148.599
C06912=1224.170,71.068,-45.981,-178.784,5.508,148.598
C06913=1224.165,71.318,-45.998,-178.781,5.509,148.598
C06914=1224.161,71.566,-46.015,-178.778,5.509,148.597
C06915=1224.155,71.816,-46.032,-178.776,5.510,148.597
C06916=1224.151,72.065,-46.050,-178.774,5.511,148.596
C06917=1224.145,72.315,-46.068,-178.771,5.511,148.595
C06918=1224.141,72.564,-46.085,-178.768,5.512,148.595
C06919=1224.136,72.814,-46.102,-178.766,5.513,148.594
C06920=1224.131,73.063,-46.120,-178.763,5.513,148.594
C06921=1224.127,73.312,-46.138,-178.761,5.514,148.593
C06922=1224.122,73.562,-46.155,-178.758,5.515,148.592
C06923=1224.117,73.811,-46.173,-178.756,5.515,148.592
C06924=1224.112,74.061,-46.190,-178.753,5.516,148.591
C06925=1224.107,74.310,-46.208,-178.751,5.517,148.590
C06926=1224.102,74.559,-46.226,-178.748,5.517,148.590
C06927=1224.097,74.808,-46.243,-178.746,5.518,148.589
C06928=1224.092,75.058,-46.261,-178.743,5.520,148.589
C06929=1224.087,75.307,-46.278,-178.740,5.520,148.588
C06930=1224.082,75.557,-46.296,-178.738,5.521,148.587
C06931=1224.078,75.805,-46.313,-178.735,5.521,148.587
C06932=1224.073,76.055,-46.331,-178.733,5.522,148.586
C06933=1224.068,76.304,-46.349,-178.730,5.523,148.586
C06934=1224.063,76.554,-46.367,-178.728,5.524,148.585
C06935=1224.058,76.803,-46.384,-178.725,5.524,148.584
C06936=1224.054,77.052,-46.401,-178.723,5.525,148.584
C06937=1224.049,77.301,-46.419,-178.720,5.526,148.583
C06938=1224.044,77.551,-46.437,-178.718,5.526,148.583
C06939=1224.039,77.800,-46.455,-178.715,5.527,148.582
C06940=1224.034,78.050,-46.473,-178.713,5.528,148.581
C06941=1224.029,78.299,-46.491,-178.710,5.529,148.581
C06942=1224.024,78.548,-46.508,-178.707,5.530,148.580
C06943=1224.019,78.798,-46.526,-178.704,5.530,148.580
C06944=1224.014,79.047,-46.543,-178.702,5.531,148.579
C06945=1224.009,79.296,-46.561,-178.700,5.532,148.578
C06946=1224.005,79.545,-46.579,-178.697,5.532,148.578
C06947=1223.999,79.795,-46.596,-178.694,5.533,148.577
C06948=1223.994,80.044,-46.614,-178.692,5.534,148.577
C06949=1223.990,80.293,-46.632,-178.690,5.535,148.576
C06950=1223.985,80.543,-46.651,-178.687,5.535,148.575
C06951=1223.980,80.792,-46.669,-178.684,5.536,148.575
C06952=1223.975,81.041,-46.687,-178.682,5.538,148.574
C06953=1223.970,81.310,-46.705,-178.679,5.538,148.574
C06954=1223.965,81.578,-46.725,-178.676,5.539,148.573
C06955=1223.959,81.846,-46.744,-178.674,5.539,148.572
C06956=1223.954,82.114,-46.763,-178.671,5.541,148.572
C06957=1223.950,82.365,-46.781,-178.668,5.541,148.571
C06958=1223.945,82.614,-46.799,-178.665,5.542,148.570
C06959=1223.940,82.863,-46.817,-178.663,5.543,148.570
C06960=1223.935,83.112,-46.835,-178.661,5.543,148.569
C06961=1223.930,83.361,-46.853,-178.658,5.544,148.569
C06962=1223.925,83.611,-46.871,-178.655,5.545,148.568
C06963=1223.920,83.860,-46.889,-178.653,5.546,148.568
C06964=1223.915,84.109,-46.907,-178.650,5.547,148.567
C06965=1223.910,84.358,-46.925,-178.647,5.548,148.566
C06966=1223.906,84.608,-46.943,-178.645,5.548,148.566
C06967=1223.901,84.857,-46.961,-178.643,5.549,148.565
C06968=1223.896,85.106,-46.979,-178.640,5.550,148.565
C06969=1223.891,85.356,-46.997,-178.637,5.550,148.564
C06970=1223.886,85.605,-47.015,-178.635,5.551,148.563
C06971=1223.881,85.854,-47.033,-178.633,5.552,148.563
C06972=1223.877,86.104,-47.051,-178.629,5.553,148.562
C06973=1223.872,86.353,-47.069,-178.627,5.554,148.562
C06974=1223.867,86.602,-47.087,-178.625,5.555,148.561
C06975=1223.862,86.852,-47.106,-178.622,5.555,148.560
C06976=1223.857,87.101,-47.124,-178.619,5.556,148.560
C06977=1223.852,87.350,-47.142,-178.617,5.557,148.559
C06978=1223.847,87.600,-47.160,-178.615,5.558,148.559
C06979=1223.843,87.849,-47.178,-178.612,5.558,148.558
C06980=1223.838,88.098,-47.196,-178.609,5.560,148.557
C06981=1223.833,88.347,-47.214,-178.607,5.560,148.557
C06982=1223.828,88.597,-47.232,-178.604,5.561,148.556
C06983=1223.824,88.846,-47.251,-178.602,5.562,148.556
C06984=1223.818,89.095,-47.270,-178.599,5.563,148.555
C06985=1223.813,89.344,-47.288,-178.597,5.563,148.555
C06986=1223.808,89.594,-47.306,-178.594,5.564,148.554
C06987=1223.803,89.843,-47.324,-178.591,5.565,148.553
C06988=1223.799,90.093,-47.342,-178.589,5.566,148.553
C06989=1223.794,90.342,-47.360,-178.586,5.567,148.552
C06990=1223.790,90.590,-47.379,-178.584,5.567,148.552
C06991=1223.784,90.840,-47.397,-178.581,5.568,148.551
C06992=1223.780,91.090,-47.416,-178.579,5.569,148.550
C06993=1223.775,91.339,-47.433,-178.576,5.570,148.550
C06994=1223.770,91.588,-47.451,-178.574,5.571,148.549
C06995=1223.765,91.837,-47.470,-178.571,5.572,148.549
C06996=1223.760,92.087,-47.489,-178.568,5.573,148.548
C06997=1223.755,92.336,-47.507,-178.566,5.573,148.547
C06998=1223.750,92.585,-47.525,-178.564,5.574,148.547
C06999=1223.746,92.834,-47.544,-178.561,5.575,148.546
C07000=1223.741,93.084,-47.563,-178.558,5.576,148.546
C07001=1223.736,93.333,-47.581,-178.556,5.577,148.545
C07002=1223.731,93.582,-47.599,-178.553,5.578,148.545
C07003=1223.727,93.832,-47.618,-178.550,5.578,148.544
C07004=1223.721,94.081,-47.636,-178.548,5.579,148.544
C07005=1223.716,94.330,-47.654,-178.546,5.580,148.543
C07006=1223.712,94.579,-47.673,-178.542,5.581,148.542
C07007=1223.707,94.829,-47.691,-178.540,5.582,148.542
C07008=1223.702,95.078,-47.710,-178.538,5.583,148.541
C07009=1223.697,95.327,-47.729,-178.535,5.583,148.541
C07010=1223.693,95.577,-47.747,-178.533,5.584,148.540
C07011=1223.687,95.826,-47.766,-178.530,5.586,148.540
C07012=1223.683,96.075,-47.784,-178.527,5.586,148.539
C07013=1223.678,96.325,-47.803,-178.525,5.587,148.538
C07014=1223.673,96.573,-47.822,-178.522,5.588,148.538
C07015=1223.668,96.823,-47.840,-178.520,5.588,148.537
C07016=1223.664,97.072,-47.858,-178.518,5.589,148.537
C07017=1223.658,97.321,-47.877,-178.514,5.591,148.536
C07018=1223.653,97.570,-47.895,-178.512,5.591,148.535
C07019=1223.649,97.820,-47.915,-178.510,5.592,148.535
C07020=1223.644,98.069,-47.933,-178.507,5.593,148.534
C07021=1223.639,98.318,-47.952,-178.504,5.594,148.534
C07022=1223.635,98.568,-47.970,-178.502,5.595,148.533
C07023=1223.629,98.817,-47.989,-178.499,5.596,148.533
C07024=1223.625,99.066,-48.007,-178.497,5.597,148.532
C07025=1223.620,99.316,-48.026,-178.494,5.598,148.532
C07026=1223.615,99.564,-48.045,-178.492,5.598,148.531
C07027=1223.611,99.814,-48.064,-178.489,5.600,148.530
C07028=1223.605,100.063,-48.083,-178.486,5.601,148.530
C07029=1223.601,100.312,-48.101,-178.484,5.601,148.529
C07030=1223.596,100.562,-48.120,-178.481,5.602,148.529
C07031=1223.591,100.811,-48.139,-178.479,5.603,148.528
C07032=1223.586,101.060,-48.157,-178.476,5.604,148.528
C07033=1223.581,101.309,-48.177,-178.473,5.605,148.527
C07034=1223.576,101.558,-48.195,-178.471,5.606,148.527
C07035=1223.572,101.808,-48.214,-178.469,5.606,148.526
C07036=1223.567,102.057,-48.232,-178.466,5.607,148.525
C07037=1223.562,102.307,-48.252,-178.463,5.609,148.525
C07038=1223.557,102.555,-48.271,-178.461,5.609,148.524
C07039=1223.552,102.805,-48.289,-178.459,5.610,148.524
C07040=1223.548,103.054,-48.308,-178.456,5.611,148.523
C07041=1223.542,103.303,-48.328,-178.453,5.612,148.523
C07042=1223.538,103.553,-48.346,-178.451,5.613,148.522
C07043=1223.533,103.802,-48.365,-178.448,5.614,148.521
C07044=1223.529,104.051,-48.384,-178.445,5.614,148.521
C07045=1223.523,104.300,-48.403,-178.443,5.615,148.520
C07046=1223.519,104.549,-48.421,-178.440,5.617,148.520
C07047=1223.514,104.799,-48.441,-178.437,5.617,148.519
C07048=1223.509,105.048,-48.459,-178.435,5.618,148.519
C07049=1223.504,105.297,-48.479,-178.433,5.619,148.518
C07050=1223.500,105.546,-48.497,-178.430,5.621,148.518
C07051=1223.494,105.796,-48.516,-178.427,5.621,148.517
C07052=1223.490,106.045,-48.535,-178.425,5.622,148.516
C07053=1223.485,106.294,-48.555,-178.423,5.623,148.516
C07054=1223.480,106.543,-48.574,-178.419,5.624,148.515
C07055=1223.475,106.793,-48.592,-178.417,5.625,148.515
C07056=1223.470,107.042,-48.612,-178.415,5.626,148.514
C07057=1223.466,107.310,-48.632,-178.412,5.627,148.514
C07058=1223.460,107.578,-48.653,-178.409,5.628,148.513
C07059=1223.455,107.847,-48.673,-178.406,5.629,148.512
C07060=1223.450,108.115,-48.694,-178.404,5.630,148.512
C07061=1223.445,108.365,-48.714,-178.401,5.631,148.511
C07062=1223.440,108.613,-48.732,-178.398,5.632,148.511
C07063=1223.435,108.864,-48.751,-178.396,5.633,148.510
C07064=1223.431,109.112,-48.770,-178.393,5.634,148.510
C07065=1223.426,109.362,-48.790,-178.391,5.635,148.509
C07066=1223.421,109.611,-48.809,-178.388,5.636,148.509
C07067=1223.417,109.860,-48.828,-178.386,5.636,148.508
C07068=1223.412,110.109,-48.848,-178.383,5.638,148.507
C07069=1223.407,110.358,-48.867,-178.380,5.639,148.507
C07070=1223.403,110.607,-48.886,-178.378,5.640,148.506
C07071=1223.397,110.857,-48.905,-178.376,5.640,148.506
C07072=1223.392,111.107,-48.924,-178.373,5.642,148.505
C07073=1223.388,111.355,-48.943,-178.370,5.643,148.505
C07074=1223.383,111.605,-48.963,-178.368,5.643,148.504
C07075=1223.377,111.854,-48.982,-178.365,5.645,148.504
C07076=1223.373,112.103,-49.002,-178.363,5.646,148.503
C07077=1223.369,112.352,-49.021,-178.360,5.646,148.502
C07078=1223.363,112.601,-49.040,-178.358,5.647,148.502
C07079=1223.359,112.851,-49.060,-178.355,5.649,148.501
C07080=1223.354,113.099,-49.078,-178.352,5.650,148.501
C07081=1223.349,113.349,-49.098,-178.350,5.650,148.500
C07082=1223.344,113.598,-49.118,-178.347,5.651,148.500
C07083=1223.339,113.847,-49.137,-178.345,5.653,148.499
C07084=1223.334,114.097,-49.156,-178.342,5.653,148.499
C07085=1223.330,114.345,-49.175,-178.340,5.654,148.498
C07086=1223.325,114.595,-49.195,-178.337,5.656,148.498
C07087=1223.320,114.845,-49.215,-178.334,5.656,148.497
C07088=1223.315,115.093,-49.234,-178.332,5.657,148.497
C07089=1223.311,115.343,-49.253,-178.329,5.658,148.496
C07090=1223.306,115.591,-49.273,-178.327,5.660,148.496
C07091=1223.301,115.841,-49.293,-178.324,5.660,148.495
C07092=1223.296,116.090,-49.312,-178.322,5.661,148.494
C07093=1223.291,116.339,-49.331,-178.319,5.663,148.494
C07094=1223.286,116.589,-49.351,-178.316,5.663,148.493
C07095=1223.282,116.838,-49.370,-178.314,5.664,148.493
C07096=1223.277,117.087,-49.389,-178.311,5.666,148.492
C07097=1223.272,117.336,-49.409,-178.309,5.667,148.492
C07098=1223.268,117.585,-49.430,-178.306,5.667,148.491
C07099=1223.262,117.834,-49.449,-178.304,5.668,148.491
C07100=1223.258,118.084,-49.468,-178.301,5.670,148.490
C07101=1223.253,118.333,-49.488,-178.299,5.671,148.490
C07102=1223.248,118.582,-49.507,-178.296,5.671,148.489
C07103=1223.244,118.831,-49.526,-178.293,5.673,148.488
C07104=1223.239,119.080,-49.547,-178.291,5.674,148.488
C07105=1223.234,119.329,-49.566,-178.288,5.674,148.487
C07106=1223.229,119.579,-49.586,-178.286,5.676,148.487
C07107=1223.224,119.828,-49.605,-178.283,5.677,148.486
C07108=1223.220,120.077,-49.626,-178.281,5.678,148.486
C07109=1223.215,120.326,-49.645,-178.278,5.679,148.485
C07110=1223.210,120.576,-49.665,-178.275,5.680,148.485
C07111=1223.205,120.825,-49.684,-178.273,5.681,148.484
C07112=1223.200,121.073,-49.704,-178.270,5.681,148.484
C07113=1223.195,121.323,-49.724,-178.268,5.683,148.483
C07114=1223.191,121.572,-49.743,-178.265,5.684,148.483
C07115=1223.187,121.821,-49.764,-178.263,5.685,148.482
C07116=1223.182,122.070,-49.783,-178.260,5.686,148.482
C07117=1223.177,122.320,-49.802,-178.258,5.687,148.481
C07118=1223.172,122.569,-49.823,-178.255,5.688,148.481
C07119=1223.168,122.818,-49.842,-178.252,5.690,148.480
C07120=1223.162,123.067,-49.862,-178.250,5.690,148.479
C07121=1223.158,123.316,-49.882,-178.248,5.691,148.479
C07122=1223.153,123.566,-49.902,-178.244,5.693,148.478
C07123=1223.149,123.815,-49.922,-178.242,5.694,148.478
C07124=1223.143,124.063,-49.941,-178.240,5.694,148.477
C07125=1223.139,124.313,-49.961,-178.237,5.696,148.477
C07126=1223.134,124.562,-49.981,-178.234,5.697,148.476
C07127=1223.129,124.812,-50.001,-178.232,5.697,148.476
C07128=1223.125,125.060,-50.022,-178.229,5.699,148.475
C07129=1223.119,125.310,-50.041,-178.226,5.700,148.475
C07130=1223.114,125.559,-50.062,-178.224,5.701,148.474
C07131=1223.110,125.808,-50.081,-178.221,5.702,148.474
C07132=1223.105,126.057,-50.102,-178.219,5.703,148.473
C07133=1223.101,126.307,-50.121,-178.216,5.705,148.473
C07134=1223.095,126.555,-50.141,-178.214,5.705,148.472
C07135=1223.091,126.804,-50.161,-178.211,5.706,148.472
C07136=1223.086,127.053,-50.181,-178.209,5.708,148.471
C07137=1223.082,127.303,-50.201,-178.206,5.709,148.471
C07138=1223.077,127.552,-50.222,-178.204,5.710,148.470
C07139=1223.072,127.802,-50.241,-178.201,5.711,148.470
C07140=1223.067,128.050,-50.261,-178.199,5.712,148.469
C07141=1223.062,128.300,-50.281,-178.196,5.713,148.469
C07142=1223.057,128.549,-50.302,-178.193,5.714,148.468
C07143=1223.053,128.798,-50.322,-178.191,5.715,148.468
C07144=1223.048,129.047,-50.342,-178.189,5.716,148.467
C07145=1223.044,129.296,-50.362,-178.185,5.717,148.467
C07146=1223.038,129.545,-50.381,-178.183,5.718,148.466
C07147=1223.034,129.794,-50.402,-178.180,5.720,148.465
C07148=1223.029,130.043,-50.423,-178.178,5.721,148.465
C07149=1223.024,130.293,-50.442,-178.175,5.721,148.464
C07150=1223.020,130.542,-50.463,-178.173,5.723,148.464
C07151=1223.015,130.791,-50.483,-178.170,5.724,148.463
C07152=1223.010,131.040,-50.503,-178.168,5.725,148.463
C07153=1223.005,131.289,-50.524,-178.165,5.726,148.462
C07154=1223.001,131.538,-50.544,-178.163,5.727,148.462
C07155=1222.996,131.787,-50.564,-178.160,5.729,148.461
C07156=1222.991,132.036,-50.584,-178.157,5.730,148.461
C07157=1222.986,132.285,-50.605,-178.155,5.730,148.460
C07158=1222.981,132.535,-50.625,-178.152,5.732,148.460
C07159=1222.977,132.784,-50.645,-178.150,5.733,148.459
C07160=1222.972,133.033,-50.665,-178.147,5.735,148.459
C07161=1222.967,133.302,-50.687,-178.144,5.735,148.458
C07162=1222.961,133.570,-50.709,-178.141,5.737,148.458
C07163=1222.957,133.840,-50.731,-178.139,5.738,148.457
C07164=1222.952,134.108,-50.753,-178.136,5.739,148.457
C07165=1222.947,134.357,-50.774,-178.134,5.740,148.456
C07166=1222.942,134.606,-50.795,-178.131,5.742,148.456
C07167=1222.937,134.856,-50.814,-178.128,5.743,148.455
C07168=1222.933,135.105,-50.835,-178.126,5.743,148.455
C07169=1222.928,135.353,-50.855,-178.123,5.745,148.454
C07170=1222.923,135.602,-50.876,-178.121,5.746,148.454
C07171=1222.918,135.851,-50.896,-178.118,5.747,148.453
C07172=1222.914,136.100,-50.916,-178.115,5.748,148.453
C07173=1222.909,136.349,-50.937,-178.113,5.750,148.452
C07174=1222.904,136.599,-50.957,-178.110,5.750,148.452
C07175=1222.899,136.848,-50.978,-178.108,5.751,148.451
C07176=1222.894,137.097,-50.998,-178.105,5.753,148.451
C07177=1222.890,137.346,-51.019,-178.103,5.754,148.450
C07178=1222.885,137.595,-51.040,-178.100,5.756,148.450
C07179=1222.880,137.844,-51.060,-178.097,5.756,148.449
C07180=1222.876,138.093,-51.080,-178.095,5.757,148.449
C07181=1222.871,138.342,-51.101,-178.092,5.759,148.448
C07182=1222.866,138.591,-51.122,-178.090,5.760,148.448
C07183=1222.861,138.841,-51.143,-178.087,5.761,148.447
C07184=1222.857,139.090,-51.163,-178.085,5.762,148.447
C07185=1222.852,139.339,-51.183,-178.081,5.764,148.446
C07186=1222.847,139.588,-51.204,-178.079,5.765,148.446
C07187=1222.842,139.837,-51.225,-178.077,5.766,148.445
C07188=1222.837,140.086,-51.246,-178.074,5.767,148.445
C07189=1222.833,140.336,-51.266,-178.072,5.768,148.444
C07190=1222.828,140.585,-51.287,-178.069,5.769,148.444
C07191=1222.824,140.834,-51.308,-178.067,5.770,148.443
C07192=1222.819,141.083,-51.328,-178.064,5.772,148.443
C07193=1222.814,141.332,-51.349,-178.061,5.773,148.442
C07194=1222.810,141.581,-51.369,-178.059,5.774,148.442
C07195=1222.805,141.830,-51.390,-178.056,5.775,148.441
C07196=1222.800,142.079,-51.411,-178.054,5.776,148.441
C07197=1222.795,142.329,-51.432,-178.051,5.778,148.440
C07198=1222.791,142.577,-51.452,-178.049,5.779,148.440
C07199=1222.786,142.826,-51.474,-178.046,5.780,148.439
C07200=1222.781,143.075,-51.494,-178.044,5.781,148.439
C07201=1222.776,143.324,-51.515,-178.041,5.783,148.439
C07202=1222.772,143.573,-51.536,-178.038,5.784,148.438
C07203=1222.767,143.823,-51.557,-178.036,5.785,148.438
C07204=1222.762,144.072,-51.578,-178.033,5.786,148.437
C07205=1222.757,144.321,-51.598,-178.031,5.787,148.437
C07206=1222.753,144.570,-51.620,-178.028,5.789,148.436
C07207=1222.748,144.819,-51.640,-178.026,5.790,148.435
C07208=1222.743,145.068,-51.661,-178.023,5.791,148.435
C07209=1222.739,145.317,-51.682,-178.020,5.792,148.434
C07210=1222.734,145.566,-51.703,-178.018,5.794,148.434
C07211=1222.730,145.816,-51.724,-178.015,5.794,148.433
C07212=1222.725,146.065,-51.745,-178.012,5.796,148.433
C07213=1222.720,146.314,-51.766,-178.010,5.797,148.433
C07214=1222.715,146.562,-51.787,-178.007,5.799,148.432
C07215=1222.710,146.812,-51.808,-178.005,5.800,148.432
C07216=1222.706,147.061,-51.828,-178.002,5.801,148.431
C07217=1222.701,147.310,-51.849,-178.000,5.802,148.431
C07218=1222.696,147.559,-51.871,-177.997,5.804,148.430
C07219=1222.692,147.808,-51.892,-177.995,5.805,148.430
C07220=1222.687,148.057,-51.913,-177.992,5.806,148.429
C07221=1222.682,148.306,-51.934,-177.989,5.807,148.429
C07222=1222.677,148.555,-51.955,-177.987,5.808,148.428
C07223=1222.672,148.804,-51.976,-177.984,5.810,148.428
C07224=1222.668,149.054,-51.998,-177.982,5.810,148.427
C07225=1222.664,149.303,-52.018,-177.979,5.812,148.427
C07226=1222.659,149.551,-52.040,-177.977,5.813,148.426
C07227=1222.653,149.800,-52.061,-177.974,5.815,148.426
C07228=1222.649,150.049,-52.081,-177.972,5.816,148.426
C07229=1222.645,150.299,-52.103,-177.969,5.817,148.425
C07230=1222.640,150.548,-52.124,-177.967,5.818,148.425
C07231=1222.635,150.797,-52.146,-177.964,5.820,148.424
C07232=1222.630,151.046,-52.166,-177.961,5.821,148.424
C07233=1222.625,151.295,-52.187,-177.959,5.822,148.423
C07234=1222.621,151.544,-52.209,-177.956,5.823,148.423
C07235=1222.616,151.793,-52.230,-177.953,5.825,148.422
C07236=1222.612,152.042,-52.251,-177.951,5.826,148.422
C07237=1222.606,152.291,-52.272,-177.948,5.827,148.421
C07238=1222.602,152.540,-52.294,-177.946,5.828,148.421
C07239=1222.597,152.790,-52.315,-177.943,5.830,148.420
C07240=1222.593,153.038,-52.336,-177.941,5.831,148.420
C07241=1222.588,153.287,-52.357,-177.938,5.833,148.419
C07242=1222.583,153.537,-52.379,-177.936,5.833,148.419
C07243=1222.578,153.785,-52.401,-177.933,5.835,148.418
C07244=1222.573,154.034,-52.422,-177.930,5.837,148.418
C07245=1222.569,154.283,-52.443,-177.928,5.838,148.417
C07246=1222.565,154.533,-52.464,-177.925,5.839,148.417
C07247=1222.560,154.781,-52.486,-177.923,5.840,148.417
C07248=1222.555,155.031,-52.507,-177.920,5.842,148.416
C07249=1222.550,155.280,-52.529,-177.918,5.843,148.416
C07250=1222.545,155.529,-52.551,-177.915,5.845,148.415
C07251=1222.540,155.778,-52.572,-177.912,5.845,148.415
C07252=1222.536,156.026,-52.593,-177.910,5.847,148.414
C07253=1222.532,156.276,-52.615,-177.908,5.848,148.414
C07254=1222.527,156.525,-52.636,-177.904,5.850,148.413
C07255=1222.522,156.773,-52.658,-177.902,5.851,148.413
C07256=1222.518,157.023,-52.680,-177.900,5.852,148.413
C07257=1222.512,157.272,-52.701,-177.897,5.853,148.412
C07258=1222.507,157.521,-52.722,-177.894,5.855,148.412
C07259=1222.503,157.770,-52.744,-177.892,5.856,148.411
C07260=1222.498,158.019,-52.765,-177.889,5.857,148.411
C07261=1222.494,158.268,-52.786,-177.886,5.859,148.410
C07262=1222.490,158.517,-52.808,-177.884,5.860,148.410
C07263=1222.485,158.766,-52.830,-177.881,5.862,148.409
C07264=1222.480,159.015,-52.851,-177.879,5.863,148.409
C07265=1222.475,159.284,-52.876,-177.876,5.864,148.408
C07266=1222.470,159.553,-52.898,-177.873,5.866,148.408
C07267=1222.465,159.823,-52.922,-177.871,5.867,148.407
C07268=1222.460,160.091,-52.946,-177.868,5.868,148.407
C07269=1222.455,160.340,-52.967,-177.865,5.870,148.406
C07270=1222.450,160.589,-52.988,-177.863,5.871,148.406
C07271=1222.445,160.839,-53.010,-177.860,5.873,148.406
C07272=1222.440,161.087,-53.032,-177.858,5.873,148.405
C07273=1222.436,161.337,-53.054,-177.855,5.875,148.405
C07274=1222.431,161.585,-53.076,-177.852,5.877,148.404
C07275=1222.426,161.834,-53.098,-177.850,5.878,148.404
C07276=1222.422,162.084,-53.119,-177.847,5.879,148.403
C07277=1222.417,162.333,-53.141,-177.845,5.880,148.403
C07278=1222.413,162.582,-53.163,-177.842,5.882,148.402
C07279=1222.408,162.831,-53.184,-177.840,5.883,148.402
C07280=1222.403,163.079,-53.206,-177.837,5.885,148.401
C07281=1222.399,163.329,-53.228,-177.834,5.887,148.401
C07282=1222.394,163.577,-53.250,-177.832,5.887,148.400
C07283=1222.390,163.826,-53.272,-177.829,5.889,148.400
C07284=1222.385,164.075,-53.293,-177.827,5.890,148.400
C07285=1222.380,164.324,-53.315,-177.824,5.892,148.399
C07286=1222.376,164.573,-53.337,-177.821,5.893,148.399
C07287=1222.371,164.822,-53.359,-177.819,5.894,148.398
C07288=1222.366,165.071,-53.381,-177.816,5.896,148.398
C07289=1222.361,165.320,-53.403,-177.814,5.897,148.397
C07290=1222.357,165.569,-53.425,-177.811,5.899,148.397
C07291=1222.352,165.818,-53.447,-177.809,5.900,148.397
C07292=1222.347,166.067,-53.469,-177.806,5.901,148.396
C07293=1222.343,166.316,-53.491,-177.803,5.903,148.396
C07294=1222.338,166.565,-53.513,-177.801,5.904,148.395
C07295=1222.333,166.814,-53.534,-177.798,5.906,148.395
C07296=1222.328,167.064,-53.557,-177.796,5.906,148.394
C07297=1222.324,167.312,-53.579,-177.793,5.908,148.394
C07298=1222.319,167.562,-53.601,-177.791,5.910,148.394
C07299=1222.315,167.810,-53.623,-177.788,5.911,148.393
C07300=1222.310,168.059,-53.645,-177.785,5.913,148.393
C07301=1222.306,168.308,-53.667,-177.783,5.914,148.392
C07302=1222.301,168.557,-53.690,-177.781,5.915,148.392
C07303=1222.296,168.806,-53.711,-177.777,5.917,148.391
C07304=1222.291,169.055,-53.733,-177.775,5.918,148.391
C07305=1222.287,169.304,-53.755,-177.773,5.920,148.391
C07306=1222.282,169.553,-53.778,-177.770,5.921,148.390
C07307=1222.278,169.802,-53.800,-177.767,5.922,148.390
C07308=1222.273,170.051,-53.822,-177.765,5.924,148.389
C07309=1222.268,170.300,-53.844,-177.763,5.925,148.389
C07310=1222.263,170.549,-53.866,-177.760,5.927,148.388
C07311=1222.259,170.798,-53.889,-177.757,5.928,148.388
